KUKA KRL program: f1_Kuka_APT216T02S16.SRC

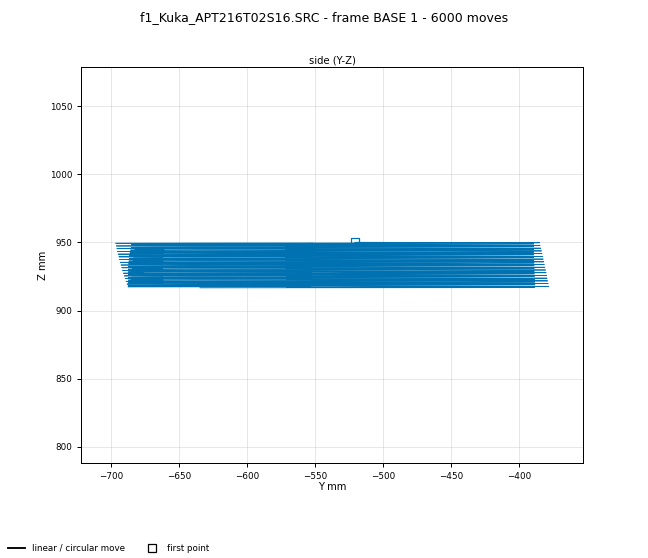
[picture p0: tool path of f1_Kuka_APT216T02S16.SRC in frame BASE 1, 6000 of 6001 moves have a stored position in this frame; points joined in program order, loops and branches not executed]
&ACCESS RVP
&REL 2
&PARAM TEMPLATE = C:\KRC\Roboter\Template\vorgabe
&PARAM EDITMASK = *
DEF f1_Kuka_APT216T02S16()


;FOLD INI;%{PE}%V3.2.0,%MKUKATPBASIS,%CINIT,%VCOMMON,%P
  ;FOLD BAS INI;%{E}%V3.2.0,%MKUKATPBASIS,%CINIT,%VINIT,%P
    GLOBAL INTERRUPT DECL 3 WHEN $STOPMESS==TRUE DO IR_STOPM ( )
    INTERRUPT ON 3
    BAS (#INITMOV,0 )
  ;ENDFOLD (BAS INI)
  ;FOLD USER INI;%{E}%V3.2.0,%MKUKATPUSER,%CINIT,%VINIT,%P
    ;Make your modifications here
  ;ENDFOLD (USER INI)
;ENDFOLD (INI)


;*** Make Null PTP Move
  PTP $pos_act

;*** Auto Load The Correct TOOL Data
  $tool=tool_data[2]

;*** Auto Load The Correct BASE Data
  $base=base_data[1]

  $ADVANCE = 5

;*** Restate Last Velocity
MMPM(30000.0)
SetRPM(8000)
LIN {X -0.232,Y -520.654,Z 950.174,A 0.000,B 0.000,C 90.000,E1 247.358} C_DIS
LIN {X 0.026,Y -518.514,Z 950.166,A 0.000,B 0.000,C 90.000,E1 245.869} C_DIS
LIN {X -0.020,Y -516.184,Z 950.158,A 0.000,B 0.000,C 90.000,E1 244.409} C_DIS
LIN {X -0.107,Y -513.864,Z 950.150,A 0.000,B 0.000,C 90.000,E1 242.948} C_DIS
LIN {X 0.234,Y -511.517,Z 950.141,A 0.000,B 0.000,C 90.000,E1 241.435} C_DIS
LIN {X 0.205,Y -509.572,Z 950.135,A 0.000,B 0.000,C 90.000,E1 240.255} C_DIS
LIN {X 0.092,Y -506.285,Z 950.125,A 0.000,B 0.000,C 90.000,E1 238.486} C_DIS
LIN {X 0.112,Y -503.056,Z 950.117,A 0.000,B 0.000,C 90.000,E1 236.993} C_DIS
LIN {X 0.178,Y -501.061,Z 950.112,A 0.000,B 0.000,C 90.000,E1 236.087} C_DIS
LIN {X -0.027,Y -497.587,Z 950.103,A 0.000,B 0.000,C 90.000,E1 234.609} C_DIS
LIN {X 0.259,Y -493.589,Z 950.093,A 0.000,B 0.000,C 90.000,E1 232.763} C_DIS
LIN {X 0.052,Y -489.488,Z 950.083,A 0.000,B 0.000,C 90.000,E1 230.964} C_DIS
LIN {X 0.021,Y -486.732,Z 950.076,A 0.000,B 0.000,C 90.000,E1 229.747} C_DIS
LIN {X -0.091,Y -482.456,Z 950.066,A 0.000,B 0.000,C 90.000,E1 227.919} C_DIS
LIN {X 0.103,Y -479.665,Z 950.059,A 0.000,B 0.000,C 90.000,E1 226.662} C_DIS
LIN {X 0.030,Y -476.272,Z 950.051,A 0.000,B 0.000,C 90.000,E1 225.121} C_DIS
LIN {X 0.084,Y -471.433,Z 950.039,A 0.000,B 0.000,C 90.000,E1 222.933} C_DIS
LIN {X -0.058,Y -467.344,Z 950.028,A 0.000,B 0.000,C 90.000,E1 221.067} C_DIS
LIN {X 0.155,Y -462.471,Z 950.016,A 0.000,B 0.000,C 90.000,E1 218.830} C_DIS
LIN {X 0.184,Y -459.007,Z 950.007,A 0.000,B 0.000,C 90.000,E1 217.237} C_DIS
LIN {X -0.125,Y -455.441,Z 949.998,A 0.000,B 0.000,C 90.000,E1 215.678} C_DIS
LIN {X 0.009,Y -449.781,Z 949.984,A 0.000,B 0.000,C 90.000,E1 213.086} C_DIS
LIN {X 0.154,Y -444.840,Z 949.971,A 0.000,B 0.000,C 90.000,E1 210.797} C_DIS
LIN {X -0.239,Y -439.153,Z 949.957,A 0.000,B 0.000,C 90.000,E1 208.231} C_DIS
LIN {X 0.100,Y -435.552,Z 949.948,A 0.000,B 0.000,C 90.000,E1 206.539} C_DIS
LIN {X -0.026,Y -431.162,Z 949.937,A 0.000,B 0.000,C 90.000,E1 204.567} C_DIS
LIN {X -0.015,Y -427.440,Z 949.927,A 0.000,B 0.000,C 90.000,E1 202.898} C_DIS
LIN {X 0.051,Y -420.044,Z 949.909,A 0.000,B 0.000,C 90.000,E1 199.523} C_DIS
LIN {X 0.037,Y -414.488,Z 949.893,A 0.000,B 0.000,C 90.000,E1 196.804} C_DIS
LIN {X 0.119,Y -411.074,Z 949.884,A 0.000,B 0.000,C 90.000,E1 195.079} C_DIS
LIN {X 0.127,Y -407.583,Z 949.874,A 0.000,B 0.000,C 90.000,E1 193.355} C_DIS
LIN {X -0.124,Y -404.196,Z 949.865,A 0.000,B 0.000,C 90.000,E1 191.658} C_DIS
LIN {X -0.050,Y -400.223,Z 949.853,A 0.000,B 0.000,C 90.000,E1 189.557} C_DIS
LIN {X -0.126,Y -396.847,Z 949.843,A 0.000,B 0.000,C 90.000,E1 187.814} C_DIS
LIN {X -0.021,Y -392.894,Z 949.832,A 0.000,B 0.000,C 90.000,E1 185.682} C_DIS
LIN {X -0.136,Y -388.562,Z 949.818,A 0.000,B 0.000,C 90.000,E1 183.212} C_DIS
LIN {X -0.091,Y -386.475,Z 949.810,A 0.000,B 0.000,C 90.000,E1 181.776} C_DIS
LIN {X 0.097,Y -385.701,Z 949.806,A 0.000,B 0.000,C 90.000,E1 181.031} C_DIS
LIN {X -0.107,Y -385.124,Z 949.802,A 0.000,B 0.000,C 90.000,E1 180.344} C_DIS
LIN {X 0.070,Y -384.918,Z 949.798,A 0.000,B 0.000,C 90.000,E1 179.599} C_DIS
LIN {X -0.140,Y -385.366,Z 949.794,A 0.000,B 0.000,C 90.000,E1 178.912} C_DIS
LIN {X 0.139,Y -385.840,Z 949.792,A 0.000,B 0.000,C 90.000,E1 178.511} C_DIS
LIN {X -0.006,Y -387.644,Z 949.788,A 0.000,B 0.000,C 90.000,E1 177.822} C_DIS
LIN {X 0.030,Y -388.934,Z 949.786,A 0.000,B 0.000,C 90.000,E1 177.478} C_DIS
LIN {X -0.113,Y -391.892,Z 949.783,A 0.000,B 0.000,C 90.000,E1 176.963} C_DIS
LIN {X 0.023,Y -394.043,Z 949.781,A 0.000,B 0.000,C 90.000,E1 176.617} C_DIS
LIN {X 0.167,Y -400.184,Z 949.778,A 0.000,B 0.000,C 90.000,E1 175.931} C_DIS
LIN {X -0.027,Y -406.077,Z 949.775,A 0.000,B 0.000,C 90.000,E1 175.412} C_DIS
LIN {X -0.026,Y -413.655,Z 949.771,A 0.000,B 0.000,C 90.000,E1 174.780} C_DIS
LIN {X 0.081,Y -421.495,Z 949.767,A 0.000,B 0.000,C 90.000,E1 174.090} C_DIS
LIN {X 0.102,Y -427.662,Z 949.764,A 0.000,B 0.000,C 90.000,E1 173.571} C_DIS
LIN {X 0.097,Y -436.825,Z 949.760,A 0.000,B 0.000,C 90.000,E1 172.761} C_DIS
LIN {X 0.074,Y -445.937,Z 949.755,A 0.000,B 0.000,C 90.000,E1 171.951} C_DIS
LIN {X -0.171,Y -455.808,Z 949.750,A 0.000,B 0.000,C 90.000,E1 171.027} C_DIS
LIN {X -0.006,Y -464.376,Z 949.745,A 0.000,B 0.000,C 90.000,E1 170.151} C_DIS
LIN {X 0.064,Y -469.840,Z 949.742,A 0.000,B 0.000,C 90.000,E1 169.567} C_DIS
LIN {X -0.010,Y -479.127,Z 949.736,A 0.000,B 0.000,C 90.000,E1 168.522} C_DIS
LIN {X -0.243,Y -484.228,Z 949.733,A 0.000,B 0.000,C 90.000,E1 167.937} C_DIS
LIN {X -0.041,Y -491.571,Z 949.728,A 0.000,B 0.000,C 90.000,E1 166.992} C_DIS
LIN {X 0.135,Y -498.521,Z 949.723,A 0.000,B 0.000,C 90.000,E1 166.061} C_DIS
LIN {X 0.092,Y -502.956,Z 949.719,A 0.000,B 0.000,C 90.000,E1 165.463} C_DIS
LIN {X 0.029,Y -509.105,Z 949.714,A 0.000,B 0.000,C 90.000,E1 164.574} C_DIS
LIN {X -0.123,Y -514.206,Z 949.710,A 0.000,B 0.000,C 90.000,E1 163.850} C_DIS
LIN {X 0.119,Y -518.896,Z 949.706,A 0.000,B 0.000,C 90.000,E1 163.087} C_DIS
LIN {X -0.265,Y -522.682,Z 949.703,A 0.000,B 0.000,C 90.000,E1 162.543} C_DIS
LIN {X 0.044,Y -529.996,Z 949.696,A 0.000,B 0.000,C 90.000,E1 161.348} C_DIS
LIN {X -0.016,Y -538.070,Z 949.689,A 0.000,B 0.000,C 90.000,E1 160.061} C_DIS
LIN {X -0.272,Y -541.475,Z 949.686,A 0.000,B 0.000,C 90.000,E1 159.518} C_DIS
LIN {X 0.310,Y -547.494,Z 949.681,A 0.000,B 0.000,C 90.000,E1 158.465} C_DIS
LIN {X 0.147,Y -554.103,Z 949.674,A 0.000,B 0.000,C 90.000,E1 157.358} C_DIS
LIN {X -0.117,Y -559.603,Z 949.669,A 0.000,B 0.000,C 90.000,E1 156.410} C_DIS
LIN {X -0.116,Y -563.343,Z 949.665,A 0.000,B 0.000,C 90.000,E1 155.717} C_DIS
LIN {X -0.015,Y -570.364,Z 949.657,A 0.000,B 0.000,C 90.000,E1 154.332} C_DIS
LIN {X -0.318,Y -576.661,Z 949.650,A 0.000,B 0.000,C 90.000,E1 152.999} C_DIS
LIN {X -0.126,Y -581.411,Z 949.644,A 0.000,B 0.000,C 90.000,E1 151.897} C_DIS
LIN {X 0.132,Y -585.685,Z 949.638,A 0.000,B 0.000,C 90.000,E1 150.795} C_DIS
LIN {X 0.172,Y -587.827,Z 949.635,A 0.000,B 0.000,C 90.000,E1 150.255} C_DIS
LIN {X -0.108,Y -592.795,Z 949.628,A 0.000,B 0.000,C 90.000,E1 148.948} C_DIS
LIN {X 0.310,Y -597.477,Z 949.620,A 0.000,B 0.000,C 90.000,E1 147.582} C_DIS
LIN {X 0.231,Y -602.930,Z 949.611,A 0.000,B 0.000,C 90.000,E1 146.008} C_DIS
LIN {X 0.070,Y -606.499,Z 949.606,A 0.000,B 0.000,C 90.000,E1 144.975} C_DIS
LIN {X 0.016,Y -611.876,Z 949.597,A 0.000,B 0.000,C 90.000,E1 143.417} C_DIS
LIN {X 0.061,Y -617.117,Z 949.588,A 0.000,B 0.000,C 90.000,E1 141.859} C_DIS
LIN {X 0.176,Y -621.563,Z 949.581,A 0.000,B 0.000,C 90.000,E1 140.561} C_DIS
LIN {X 0.025,Y -632.173,Z 949.564,A 0.000,B 0.000,C 90.000,E1 137.514} C_DIS
LIN {X 0.159,Y -634.999,Z 949.560,A 0.000,B 0.000,C 90.000,E1 136.743} C_DIS
LIN {X 0.041,Y -640.541,Z 949.551,A 0.000,B 0.000,C 90.000,E1 135.243} C_DIS
LIN {X 0.033,Y -646.038,Z 949.543,A 0.000,B 0.000,C 90.000,E1 133.743} C_DIS
LIN {X 0.086,Y -652.493,Z 949.533,A 0.000,B 0.000,C 90.000,E1 132.000} C_DIS
LIN {X -0.171,Y -658.949,Z 949.524,A 0.000,B 0.000,C 90.000,E1 130.297} C_DIS
LIN {X -0.190,Y -664.562,Z 949.516,A 0.000,B 0.000,C 90.000,E1 128.830} C_DIS
LIN {X -0.097,Y -670.115,Z 949.508,A 0.000,B 0.000,C 90.000,E1 127.363} C_DIS
LIN {X 0.112,Y -673.593,Z 949.502,A 0.000,B 0.000,C 90.000,E1 126.377} C_DIS
LIN {X -0.178,Y -676.931,Z 949.497,A 0.000,B 0.000,C 90.000,E1 125.438} C_DIS
LIN {X 0.289,Y -680.765,Z 949.490,A 0.000,B 0.000,C 90.000,E1 124.199} C_DIS
LIN {X -0.119,Y -684.239,Z 949.484,A 0.000,B 0.000,C 90.000,E1 123.038} C_DIS
LIN {X -0.102,Y -686.803,Z 949.478,A 0.000,B 0.000,C 90.000,E1 122.084} C_DIS
LIN {X -0.055,Y -689.089,Z 949.473,A 0.000,B 0.000,C 90.000,E1 121.131} C_DIS
LIN {X -0.200,Y -690.201,Z 949.470,A 0.000,B 0.000,C 90.000,E1 120.669} C_DIS
LIN {X -0.125,Y -692.059,Z 949.465,A 0.000,B 0.000,C 90.000,E1 119.716} C_DIS
LIN {X 0.229,Y -693.569,Z 949.460,A 0.000,B 0.000,C 90.000,E1 118.743} C_DIS
LIN {X 0.031,Y -694.577,Z 949.456,A 0.000,B 0.000,C 90.000,E1 118.052} C_DIS
LIN {X -0.189,Y -695.499,Z 949.451,A 0.000,B 0.000,C 90.000,E1 117.129} C_DIS
LIN {X -0.098,Y -696.065,Z 949.445,A 0.000,B 0.000,C 90.000,E1 116.181} C_DIS
LIN {X -0.364,Y -696.413,Z 949.439,A 0.000,B 0.000,C 90.000,E1 115.027} C_DIS
LIN {X 0.119,Y -696.392,Z 949.435,A 0.000,B 0.000,C 90.000,E1 114.283} C_DIS
LIN {X -0.005,Y -696.185,Z 949.432,A 0.000,B 0.000,C 90.000,E1 113.823} C_DIS
LIN {X 0.224,Y -695.279,Z 949.430,A 0.000,B 0.000,C 90.000,E1 113.334} C_DIS
LIN {X -0.165,Y -694.668,Z 949.428,A 0.000,B 0.000,C 90.000,E1 113.131} C_DIS
LIN {X -0.066,Y -692.739,Z 949.427,A 0.000,B 0.000,C 90.000,E1 112.770} C_DIS
LIN {X 0.174,Y -691.341,Z 949.425,A 0.000,B 0.000,C 90.000,E1 112.514} C_DIS
LIN {X 0.029,Y -690.332,Z 949.425,A 0.000,B 0.000,C 90.000,E1 112.408} C_DIS
LIN {X 0.145,Y -688.808,Z 949.424,A 0.000,B 0.000,C 90.000,E1 112.280} C_DIS
LIN {X -0.266,Y -683.650,Z 949.422,A 0.000,B 0.000,C 90.000,E1 112.025} C_DIS
LIN {X -0.132,Y -681.695,Z 949.422,A 0.000,B 0.000,C 90.000,E1 111.897} C_DIS
LIN {X -0.112,Y -676.345,Z 949.421,A 0.000,B 0.000,C 90.000,E1 111.716} C_DIS
LIN {X -0.005,Y -673.275,Z 949.420,A 0.000,B 0.000,C 90.000,E1 111.663} C_DIS
LIN {X 0.233,Y -667.551,Z 949.420,A 0.000,B 0.000,C 90.000,E1 111.589} C_DIS
LIN {X 0.175,Y -634.091,Z 949.420,A 0.000,B 0.000,C 90.000,E1 111.589} C_DIS
LIN {X 0.193,Y -629.702,Z 949.420,A 0.000,B 0.000,C 90.000,E1 111.535} C_DIS
LIN {X 0.223,Y -622.529,Z 949.419,A 0.000,B 0.000,C 90.000,E1 111.408} C_DIS
LIN {X 0.174,Y -615.532,Z 949.418,A 0.000,B 0.000,C 90.000,E1 111.227} C_DIS
LIN {X 0.223,Y -608.532,Z 949.417,A 0.000,B 0.000,C 90.000,E1 110.972} C_DIS
LIN {X -0.059,Y -600.335,Z 949.414,A 0.000,B 0.000,C 90.000,E1 110.610} C_DIS
LIN {X 0.310,Y -593.030,Z 949.412,A 0.000,B 0.000,C 90.000,E1 110.120} C_DIS
LIN {X -0.139,Y -577.483,Z 949.406,A 0.000,B 0.000,C 90.000,E1 109.033} C_DIS
LIN {X -0.162,Y -574.078,Z 949.405,A 0.000,B 0.000,C 90.000,E1 108.833} C_DIS
LIN {X -0.024,Y -569.119,Z 949.403,A 0.000,B 0.000,C 90.000,E1 108.544} C_DIS
LIN {X -0.086,Y -563.607,Z 949.402,A 0.000,B 0.000,C 90.000,E1 108.290} C_DIS
LIN {X 0.267,Y -555.303,Z 949.399,A 0.000,B 0.000,C 90.000,E1 107.873} C_DIS
LIN {X 0.222,Y -553.260,Z 949.399,A 0.000,B 0.000,C 90.000,E1 107.764} C_DIS
LIN {X -0.084,Y -551.662,Z 949.398,A 0.000,B 0.000,C 90.000,E1 107.638} C_DIS
LIN {X -0.137,Y -551.620,Z 949.398,A 0.000,B 0.000,C 90.000,E1 107.638} C_DIS
LIN {X -0.215,Y -551.221,Z 949.397,A 0.000,B 0.000,C 90.000,E1 107.457} C_DIS
LIN {X -0.144,Y -551.117,Z 949.395,A 0.000,B 0.000,C 90.000,E1 107.149} C_DIS
LIN {X 0.261,Y -551.695,Z 949.386,A 0.000,B 0.000,C 90.000,E1 105.426} C_DIS
LIN {X -0.161,Y -552.767,Z 949.373,A 0.000,B 0.000,C 90.000,E1 103.231} C_DIS
LIN {X -0.023,Y -554.814,Z 949.358,A 0.000,B 0.000,C 90.000,E1 100.423} C_DIS
LIN {X -0.026,Y -556.065,Z 949.350,A 0.000,B 0.000,C 90.000,E1 99.029} C_DIS
LIN {X -0.086,Y -557.277,Z 949.342,A 0.000,B 0.000,C 90.000,E1 97.644} C_DIS
LIN {X -0.187,Y -558.194,Z 949.336,A 0.000,B 0.000,C 90.000,E1 96.543} C_DIS
LIN {X 0.212,Y -558.934,Z 949.330,A 0.000,B 0.000,C 90.000,E1 95.391} C_DIS
LIN {X 0.018,Y -559.641,Z 949.324,A 0.000,B 0.000,C 90.000,E1 94.302} C_DIS
LIN {X 0.054,Y -560.601,Z 949.315,A 0.000,B 0.000,C 90.000,E1 92.636} C_DIS
LIN {X -0.113,Y -561.108,Z 949.309,A 0.000,B 0.000,C 90.000,E1 91.547} C_DIS
LIN {X -0.190,Y -561.700,Z 949.301,A 0.000,B 0.000,C 90.000,E1 90.172} C_DIS
LIN {X 0.207,Y -562.043,Z 949.295,A 0.000,B 0.000,C 90.000,E1 89.026} C_DIS
LIN {X 0.161,Y -562.350,Z 949.287,A 0.000,B 0.000,C 90.000,E1 87.650} C_DIS
LIN {X 0.120,Y -562.635,Z 949.279,A 0.000,B 0.000,C 90.000,E1 86.274} C_DIS
LIN {X 0.210,Y -562.883,Z 949.270,A 0.000,B 0.000,C 90.000,E1 84.609} C_DIS
LIN {X -0.140,Y -563.149,Z 949.261,A 0.000,B 0.000,C 90.000,E1 82.989} C_DIS
LIN {X -0.072,Y -563.754,Z 949.247,A 0.000,B 0.000,C 90.000,E1 80.500} C_DIS
LIN {X 0.032,Y -564.679,Z 949.235,A 0.000,B 0.000,C 90.000,E1 78.285} C_DIS
LIN {X -0.287,Y -565.934,Z 949.223,A 0.000,B 0.000,C 90.000,E1 76.117} C_DIS
LIN {X -0.089,Y -566.976,Z 949.214,A 0.000,B 0.000,C 90.000,E1 74.448} C_DIS
LIN {X 0.136,Y -568.043,Z 949.204,A 0.000,B 0.000,C 90.000,E1 72.779} C_DIS
LIN {X 0.207,Y -568.808,Z 949.197,A 0.000,B 0.000,C 90.000,E1 71.402} C_DIS
LIN {X -0.066,Y -569.546,Z 949.189,A 0.000,B 0.000,C 90.000,E1 70.061} C_DIS
LIN {X 0.020,Y -570.119,Z 949.180,A 0.000,B 0.000,C 90.000,E1 68.411} C_DIS
LIN {X -0.202,Y -570.590,Z 949.171,A 0.000,B 0.000,C 90.000,E1 66.794} C_DIS
LIN {X 0.170,Y -571.025,Z 949.160,A 0.000,B 0.000,C 90.000,E1 64.845} C_DIS
LIN {X 0.192,Y -571.266,Z 949.151,A 0.000,B 0.000,C 90.000,E1 63.204} C_DIS
LIN {X 0.125,Y -571.435,Z 949.144,A 0.000,B 0.000,C 90.000,E1 61.847} C_DIS
LIN {X 0.165,Y -571.468,Z 949.135,A 0.000,B 0.000,C 90.000,E1 60.205} C_DIS
LIN {X 0.008,Y -571.634,Z 949.126,A 0.000,B 0.000,C 90.000,E1 58.584} C_DIS
LIN {X -0.266,Y -571.503,Z 949.118,A 0.000,B 0.000,C 90.000,E1 57.248} C_DIS
LIN {X -0.244,Y -571.139,Z 949.110,A 0.000,B 0.000,C 90.000,E1 55.881} C_DIS
LIN {X 0.092,Y -570.671,Z 949.103,A 0.000,B 0.000,C 90.000,E1 54.482} C_DIS
LIN {X 0.357,Y -570.473,Z 949.100,A 0.000,B 0.000,C 90.000,E1 53.909} C_DIS
LIN {X -0.045,Y -569.986,Z 949.095,A 0.000,B 0.000,C 90.000,E1 53.130} C_DIS
LIN {X 0.024,Y -569.081,Z 949.089,A 0.000,B 0.000,C 90.000,E1 52.029} C_DIS
LIN {X 0.085,Y -568.018,Z 949.083,A 0.000,B 0.000,C 90.000,E1 50.928} C_DIS
LIN {X 0.010,Y -567.101,Z 949.078,A 0.000,B 0.000,C 90.000,E1 50.114} C_DIS
LIN {X -0.077,Y -566.046,Z 949.074,A 0.000,B 0.000,C 90.000,E1 49.299} C_DIS
LIN {X -0.181,Y -564.794,Z 949.069,A 0.000,B 0.000,C 90.000,E1 48.485} C_DIS
LIN {X -0.248,Y -562.711,Z 949.063,A 0.000,B 0.000,C 90.000,E1 47.391} C_DIS
LIN {X -0.098,Y -561.646,Z 949.060,A 0.000,B 0.000,C 90.000,E1 46.824} C_DIS
LIN {X 0.122,Y -559.750,Z 949.056,A 0.000,B 0.000,C 90.000,E1 45.972} C_DIS
LIN {X -0.081,Y -557.570,Z 949.051,A 0.000,B 0.000,C 90.000,E1 45.162} C_DIS
LIN {X 0.034,Y -556.031,Z 949.048,A 0.000,B 0.000,C 90.000,E1 44.595} C_DIS
LIN {X -0.207,Y -553.337,Z 949.043,A 0.000,B 0.000,C 90.000,E1 43.785} C_DIS
LIN {X -0.125,Y -551.495,Z 949.040,A 0.000,B 0.000,C 90.000,E1 43.218} C_DIS
LIN {X -0.017,Y -548.288,Z 949.035,A 0.000,B 0.000,C 90.000,E1 42.366} C_DIS
LIN {X 0.056,Y -544.757,Z 949.031,A 0.000,B 0.000,C 90.000,E1 41.515} C_DIS
LIN {X 0.281,Y -542.809,Z 949.028,A 0.000,B 0.000,C 90.000,E1 41.067} C_DIS
LIN {X -0.064,Y -538.565,Z 949.024,A 0.000,B 0.000,C 90.000,E1 40.253} C_DIS
LIN {X -0.279,Y -534.725,Z 949.020,A 0.000,B 0.000,C 90.000,E1 39.564} C_DIS
LIN {X 0.043,Y -529.767,Z 949.015,A 0.000,B 0.000,C 90.000,E1 38.669} C_DIS
LIN {X 0.122,Y -523.679,Z 949.009,A 0.000,B 0.000,C 90.000,E1 37.649} C_DIS
LIN {X 0.041,Y -520.035,Z 949.006,A 0.000,B 0.000,C 90.000,E1 37.076} C_DIS
LIN {X -0.312,Y -513.139,Z 949.000,A 0.000,B 0.000,C 90.000,E1 36.091} C_DIS
LIN {X 0.055,Y -507.914,Z 948.996,A 0.000,B 0.000,C 90.000,E1 35.311} C_DIS
LIN {X -0.138,Y -503.436,Z 948.993,A 0.000,B 0.000,C 90.000,E1 34.739} C_DIS
LIN {X -0.031,Y -499.916,Z 948.990,A 0.000,B 0.000,C 90.000,E1 34.278} C_DIS
LIN {X -0.079,Y -496.182,Z 948.988,A 0.000,B 0.000,C 90.000,E1 33.833} C_DIS
LIN {X -0.167,Y -488.144,Z 948.983,A 0.000,B 0.000,C 90.000,E1 32.959} C_DIS
LIN {X 0.054,Y -481.171,Z 948.979,A 0.000,B 0.000,C 90.000,E1 32.212} C_DIS
LIN {X -0.140,Y -475.423,Z 948.976,A 0.000,B 0.000,C 90.000,E1 31.671} C_DIS
LIN {X -0.059,Y -466.585,Z 948.971,A 0.000,B 0.000,C 90.000,E1 30.846} C_DIS
LIN {X -0.078,Y -459.131,Z 948.968,A 0.000,B 0.000,C 90.000,E1 30.178} C_DIS
LIN {X -0.255,Y -448.516,Z 948.963,A 0.000,B 0.000,C 90.000,E1 29.283} C_DIS
LIN {X -0.056,Y -428.627,Z 948.953,A 0.000,B 0.000,C 90.000,E1 27.564} C_DIS
LIN {X -0.085,Y -412.114,Z 948.945,A 0.000,B 0.000,C 90.000,E1 26.052} C_DIS
LIN {X 0.032,Y -400.392,Z 948.938,A 0.000,B 0.000,C 90.000,E1 24.847} C_DIS
LIN {X 0.149,Y -397.529,Z 948.936,A 0.000,B 0.000,C 90.000,E1 24.515} C_DIS
LIN {X -0.027,Y -394.399,Z 948.934,A 0.000,B 0.000,C 90.000,E1 24.131} C_DIS
LIN {X -0.152,Y -392.235,Z 948.932,A 0.000,B 0.000,C 90.000,E1 23.770} C_DIS
LIN {X 0.028,Y -391.305,Z 948.931,A 0.000,B 0.000,C 90.000,E1 23.567} C_DIS
LIN {X 0.111,Y -389.845,Z 948.928,A 0.000,B 0.000,C 90.000,E1 23.025} C_DIS
LIN {X -0.029,Y -389.162,Z 948.924,A 0.000,B 0.000,C 90.000,E1 22.333} C_DIS
LIN {X 0.201,Y -389.528,Z 948.919,A 0.000,B 0.000,C 90.000,E1 21.408} C_DIS
LIN {X 0.076,Y -393.067,Z 948.897,A 0.000,B 0.000,C 90.000,E1 17.511} C_DIS
LIN {X -0.181,Y -396.430,Z 948.882,A 0.000,B 0.000,C 90.000,E1 14.717} C_DIS
LIN {X -0.107,Y -399.795,Z 948.868,A 0.000,B 0.000,C 90.000,E1 12.243} C_DIS
LIN {X -0.097,Y -404.793,Z 948.851,A 0.000,B 0.000,C 90.000,E1 9.095} C_DIS
LIN {X -0.041,Y -410.390,Z 948.833,A 0.000,B 0.000,C 90.000,E1 5.967} C_DIS
LIN {X 0.057,Y -417.434,Z 948.814,A 0.000,B 0.000,C 90.000,E1 2.522} C_DIS
LIN {X 0.208,Y -424.749,Z 948.797,A 0.000,B 0.000,C 90.000,E1 359.427} C_DIS
LIN {X -0.167,Y -425.696,Z 948.795,A 0.000,B 0.000,C 90.000,E1 359.141} C_DIS
LIN {X -0.058,Y -428.393,Z 948.791,A 0.000,B 0.000,C 90.000,E1 358.453} C_DIS
LIN {X 0.090,Y -429.543,Z 948.790,A 0.000,B 0.000,C 90.000,E1 358.224} C_DIS
LIN {X 0.092,Y -431.486,Z 948.789,A 0.000,B 0.000,C 90.000,E1 357.936} C_DIS
LIN {X 0.216,Y -435.092,Z 948.786,A 0.000,B 0.000,C 90.000,E1 357.535} C_DIS
LIN {X 0.188,Y -440.022,Z 948.785,A 0.000,B 0.000,C 90.000,E1 357.192} C_DIS
LIN {X 0.066,Y -458.415,Z 948.779,A 0.000,B 0.000,C 90.000,E1 356.274} C_DIS
LIN {X -0.181,Y -466.700,Z 948.777,A 0.000,B 0.000,C 90.000,E1 355.869} C_DIS
LIN {X 0.094,Y -480.168,Z 948.773,A 0.000,B 0.000,C 90.000,E1 355.122} C_DIS
LIN {X 0.084,Y -491.926,Z 948.769,A 0.000,B 0.000,C 90.000,E1 354.489} C_DIS
LIN {X -0.062,Y -498.505,Z 948.768,A 0.000,B 0.000,C 90.000,E1 354.147} C_DIS
LIN {X 0.115,Y -507.951,Z 948.764,A 0.000,B 0.000,C 90.000,E1 353.571} C_DIS
LIN {X -0.046,Y -517.568,Z 948.761,A 0.000,B 0.000,C 90.000,E1 352.996} C_DIS
LIN {X 0.144,Y -526.710,Z 948.758,A 0.000,B 0.000,C 90.000,E1 352.356} C_DIS
LIN {X -0.198,Y -534.129,Z 948.755,A 0.000,B 0.000,C 90.000,E1 351.837} C_DIS
LIN {X -0.212,Y -541.363,Z 948.751,A 0.000,B 0.000,C 90.000,E1 351.254} C_DIS
LIN {X -0.050,Y -548.207,Z 948.748,A 0.000,B 0.000,C 90.000,E1 350.622} C_DIS
LIN {X -0.234,Y -554.623,Z 948.744,A 0.000,B 0.000,C 90.000,E1 349.982} C_DIS
LIN {X 0.135,Y -559.615,Z 948.741,A 0.000,B 0.000,C 90.000,E1 349.398} C_DIS
LIN {X 0.181,Y -565.330,Z 948.737,A 0.000,B 0.000,C 90.000,E1 348.701} C_DIS
LIN {X -0.037,Y -569.568,Z 948.734,A 0.000,B 0.000,C 90.000,E1 348.173} C_DIS
LIN {X 0.211,Y -574.517,Z 948.731,A 0.000,B 0.000,C 90.000,E1 347.465} C_DIS
LIN {X 0.273,Y -579.999,Z 948.726,A 0.000,B 0.000,C 90.000,E1 346.645} C_DIS
LIN {X 0.058,Y -586.520,Z 948.720,A 0.000,B 0.000,C 90.000,E1 345.589} C_DIS
LIN {X 0.307,Y -591.809,Z 948.715,A 0.000,B 0.000,C 90.000,E1 344.629} C_DIS
LIN {X -0.106,Y -596.683,Z 948.710,A 0.000,B 0.000,C 90.000,E1 343.740} C_DIS
LIN {X 0.047,Y -601.896,Z 948.704,A 0.000,B 0.000,C 90.000,E1 342.670} C_DIS
LIN {X 0.179,Y -608.028,Z 948.697,A 0.000,B 0.000,C 90.000,E1 341.348} C_DIS
LIN {X 0.085,Y -612.604,Z 948.691,A 0.000,B 0.000,C 90.000,E1 340.315} C_DIS
LIN {X 0.013,Y -617.926,Z 948.684,A 0.000,B 0.000,C 90.000,E1 339.028} C_DIS
LIN {X 0.275,Y -621.863,Z 948.678,A 0.000,B 0.000,C 90.000,E1 337.975} C_DIS
LIN {X 0.019,Y -625.619,Z 948.672,A 0.000,B 0.000,C 90.000,E1 336.975} C_DIS
LIN {X -0.165,Y -629.912,Z 948.665,A 0.000,B 0.000,C 90.000,E1 335.717} C_DIS
LIN {X 0.292,Y -633.837,Z 948.658,A 0.000,B 0.000,C 90.000,E1 334.409} C_DIS
LIN {X -0.057,Y -637.521,Z 948.651,A 0.000,B 0.000,C 90.000,E1 333.179} C_DIS
LIN {X 0.166,Y -640.207,Z 948.645,A 0.000,B 0.000,C 90.000,E1 332.153} C_DIS
LIN {X -0.146,Y -642.621,Z 948.640,A 0.000,B 0.000,C 90.000,E1 331.179} C_DIS
LIN {X -0.040,Y -645.468,Z 948.633,A 0.000,B 0.000,C 90.000,E1 329.921} C_DIS
LIN {X 0.114,Y -648.016,Z 948.626,A 0.000,B 0.000,C 90.000,E1 328.663} C_DIS
LIN {X -0.252,Y -650.147,Z 948.619,A 0.000,B 0.000,C 90.000,E1 327.454} C_DIS
LIN {X 0.229,Y -651.668,Z 948.614,A 0.000,B 0.000,C 90.000,E1 326.421} C_DIS
LIN {X 0.272,Y -653.310,Z 948.607,A 0.000,B 0.000,C 90.000,E1 325.182} C_DIS
LIN {X -0.195,Y -654.159,Z 948.603,A 0.000,B 0.000,C 90.000,E1 324.482} C_DIS
LIN {X -0.201,Y -655.114,Z 948.597,A 0.000,B 0.000,C 90.000,E1 323.497} C_DIS
LIN {X 0.204,Y -656.376,Z 948.589,A 0.000,B 0.000,C 90.000,E1 321.984} C_DIS
LIN {X 0.074,Y -657.682,Z 948.579,A 0.000,B 0.000,C 90.000,E1 320.275} C_DIS
LIN {X -0.029,Y -658.532,Z 948.573,A 0.000,B 0.000,C 90.000,E1 319.057} C_DIS
LIN {X -0.226,Y -660.444,Z 948.558,A 0.000,B 0.000,C 90.000,E1 316.377} C_DIS
LIN {X -0.304,Y -661.245,Z 948.552,A 0.000,B 0.000,C 90.000,E1 315.405} C_DIS
LIN {X 0.044,Y -663.106,Z 948.540,A 0.000,B 0.000,C 90.000,E1 313.176} C_DIS
LIN {X 0.021,Y -664.458,Z 948.532,A 0.000,B 0.000,C 90.000,E1 311.714} C_DIS
LIN {X 0.035,Y -665.578,Z 948.525,A 0.000,B 0.000,C 90.000,E1 310.496} C_DIS
LIN {X 0.059,Y -666.560,Z 948.518,A 0.000,B 0.000,C 90.000,E1 309.277} C_DIS
LIN {X -0.333,Y -667.496,Z 948.512,A 0.000,B 0.000,C 90.000,E1 308.096} C_DIS
LIN {X -0.251,Y -667.873,Z 948.509,A 0.000,B 0.000,C 90.000,E1 307.604} C_DIS
LIN {X -0.097,Y -668.375,Z 948.502,A 0.000,B 0.000,C 90.000,E1 306.377} C_DIS
LIN {X -0.235,Y -668.877,Z 948.493,A 0.000,B 0.000,C 90.000,E1 304.692} C_DIS
LIN {X 0.188,Y -669.527,Z 948.483,A 0.000,B 0.000,C 90.000,E1 302.959} C_DIS
LIN {X 0.253,Y -670.367,Z 948.474,A 0.000,B 0.000,C 90.000,E1 301.258} C_DIS
LIN {X 0.345,Y -674.131,Z 948.452,A 0.000,B 0.000,C 90.000,E1 297.385} C_DIS
LIN {X -0.410,Y -677.717,Z 948.440,A 0.000,B 0.000,C 90.000,E1 295.283} C_DIS
LIN {X -0.346,Y -679.725,Z 948.434,A 0.000,B 0.000,C 90.000,E1 294.079} C_DIS
LIN {X -0.032,Y -680.838,Z 948.430,A 0.000,B 0.000,C 90.000,E1 293.334} C_DIS
LIN {X -0.331,Y -681.524,Z 948.426,A 0.000,B 0.000,C 90.000,E1 292.642} C_DIS
LIN {X -0.194,Y -681.362,Z 948.423,A 0.000,B 0.000,C 90.000,E1 292.153} C_DIS
LIN {X 0.002,Y -681.134,Z 948.422,A 0.000,B 0.000,C 90.000,E1 291.897} C_DIS
LIN {X -0.056,Y -680.338,Z 948.420,A 0.000,B 0.000,C 90.000,E1 291.663} C_DIS
LIN {X 0.080,Y -678.053,Z 948.418,A 0.000,B 0.000,C 90.000,E1 291.173} C_DIS
LIN {X 0.172,Y -677.053,Z 948.417,A 0.000,B 0.000,C 90.000,E1 291.046} C_DIS
LIN {X -0.223,Y -674.434,Z 948.416,A 0.000,B 0.000,C 90.000,E1 290.844} C_DIS
LIN {X -0.077,Y -671.639,Z 948.414,A 0.000,B 0.000,C 90.000,E1 290.610} C_DIS
LIN {X -0.020,Y -666.907,Z 948.413,A 0.000,B 0.000,C 90.000,E1 290.301} C_DIS
LIN {X 0.227,Y -661.860,Z 948.411,A 0.000,B 0.000,C 90.000,E1 289.939} C_DIS
LIN {X -0.028,Y -660.825,Z 948.411,A 0.000,B 0.000,C 90.000,E1 289.885} C_DIS
LIN {X -0.096,Y -660.785,Z 948.410,A 0.000,B 0.000,C 90.000,E1 289.885} C_DIS
LIN {X 0.292,Y -660.270,Z 948.410,A 0.000,B 0.000,C 90.000,E1 289.758} C_DIS
LIN {X 0.225,Y -660.259,Z 948.410,A 0.000,B 0.000,C 90.000,E1 289.758} C_DIS
LIN {X 0.102,Y -660.344,Z 948.409,A 0.000,B 0.000,C 90.000,E1 289.523} C_DIS
LIN {X 0.125,Y -660.794,Z 948.408,A 0.000,B 0.000,C 90.000,E1 289.341} C_DIS
LIN {X 0.289,Y -662.012,Z 948.406,A 0.000,B 0.000,C 90.000,E1 288.960} C_DIS
LIN {X 0.086,Y -669.194,Z 948.398,A 0.000,B 0.000,C 90.000,E1 287.638} C_DIS
LIN {X -0.064,Y -671.729,Z 948.395,A 0.000,B 0.000,C 90.000,E1 287.166} C_DIS
LIN {X -0.064,Y -674.896,Z 948.391,A 0.000,B 0.000,C 90.000,E1 286.441} C_DIS
LIN {X -0.043,Y -677.464,Z 948.387,A 0.000,B 0.000,C 90.000,E1 285.717} C_DIS
LIN {X -0.138,Y -678.887,Z 948.385,A 0.000,B 0.000,C 90.000,E1 285.245} C_DIS
LIN {X -0.262,Y -680.604,Z 948.381,A 0.000,B 0.000,C 90.000,E1 284.537} C_DIS
LIN {X 0.296,Y -681.962,Z 948.377,A 0.000,B 0.000,C 90.000,E1 283.772} C_DIS
LIN {X 0.206,Y -683.143,Z 948.373,A 0.000,B 0.000,C 90.000,E1 283.063} C_DIS
LIN {X 0.124,Y -684.038,Z 948.369,A 0.000,B 0.000,C 90.000,E1 282.355} C_DIS
LIN {X -0.095,Y -684.630,Z 948.365,A 0.000,B 0.000,C 90.000,E1 281.658} C_DIS
LIN {X -0.144,Y -684.816,Z 948.362,A 0.000,B 0.000,C 90.000,E1 281.186} C_DIS
LIN {X -0.197,Y -684.693,Z 948.359,A 0.000,B 0.000,C 90.000,E1 280.715} C_DIS
LIN {X 0.297,Y -684.272,Z 948.357,A 0.000,B 0.000,C 90.000,E1 280.197} C_DIS
LIN {X 0.236,Y -683.453,Z 948.354,A 0.000,B 0.000,C 90.000,E1 279.726} C_DIS
LIN {X 0.054,Y -682.344,Z 948.352,A 0.000,B 0.000,C 90.000,E1 279.265} C_DIS
LIN {X 0.016,Y -681.735,Z 948.350,A 0.000,B 0.000,C 90.000,E1 279.029} C_DIS
LIN {X -0.173,Y -680.105,Z 948.348,A 0.000,B 0.000,C 90.000,E1 278.568} C_DIS
LIN {X 0.247,Y -677.032,Z 948.344,A 0.000,B 0.000,C 90.000,E1 277.814} C_DIS
LIN {X -0.122,Y -673.513,Z 948.340,A 0.000,B 0.000,C 90.000,E1 277.125} C_DIS
LIN {X -0.274,Y -671.594,Z 948.338,A 0.000,B 0.000,C 90.000,E1 276.777} C_DIS
LIN {X 0.143,Y -668.794,Z 948.335,A 0.000,B 0.000,C 90.000,E1 276.258} C_DIS
LIN {X -0.125,Y -665.751,Z 948.332,A 0.000,B 0.000,C 90.000,E1 275.796} C_DIS
LIN {X 0.158,Y -661.292,Z 948.329,A 0.000,B 0.000,C 90.000,E1 275.163} C_DIS
LIN {X -0.119,Y -658.439,Z 948.327,A 0.000,B 0.000,C 90.000,E1 274.821} C_DIS
LIN {X 0.001,Y -651.781,Z 948.323,A 0.000,B 0.000,C 90.000,E1 274.073} C_DIS
LIN {X 0.272,Y -647.055,Z 948.320,A 0.000,B 0.000,C 90.000,E1 273.555} C_DIS
LIN {X -0.012,Y -642.044,Z 948.317,A 0.000,B 0.000,C 90.000,E1 273.094} C_DIS
LIN {X -0.136,Y -636.787,Z 948.315,A 0.000,B 0.000,C 90.000,E1 272.636} C_DIS
LIN {X -0.096,Y -631.333,Z 948.312,A 0.000,B 0.000,C 90.000,E1 272.178} C_DIS
LIN {X -0.280,Y -624.030,Z 948.309,A 0.000,B 0.000,C 90.000,E1 271.661} C_DIS
LIN {X -0.077,Y -616.380,Z 948.306,A 0.000,B 0.000,C 90.000,E1 271.146} C_DIS
LIN {X 0.116,Y -610.051,Z 948.304,A 0.000,B 0.000,C 90.000,E1 270.745} C_DIS
LIN {X -0.017,Y -603.473,Z 948.302,A 0.000,B 0.000,C 90.000,E1 270.401} C_DIS
LIN {X -0.235,Y -598.439,Z 948.301,A 0.000,B 0.000,C 90.000,E1 270.172} C_DIS
LIN {X 0.160,Y -591.399,Z 948.299,A 0.000,B 0.000,C 90.000,E1 269.828} C_DIS
LIN {X 0.278,Y -584.013,Z 948.298,A 0.000,B 0.000,C 90.000,E1 269.542} C_DIS
LIN {X 0.234,Y -578.151,Z 948.297,A 0.000,B 0.000,C 90.000,E1 269.370} C_DIS
LIN {X 0.080,Y -570.455,Z 948.296,A 0.000,B 0.000,C 90.000,E1 269.198} C_DIS
LIN {X 0.056,Y -564.645,Z 948.295,A 0.000,B 0.000,C 90.000,E1 269.083} C_DIS
LIN {X -0.096,Y -558.396,Z 948.295,A 0.000,B 0.000,C 90.000,E1 269.026} C_DIS
LIN {X 0.014,Y -550.975,Z 948.294,A 0.000,B 0.000,C 90.000,E1 268.969} C_DIS
LIN {X 0.200,Y -548.037,Z 948.294,A 0.000,B 0.000,C 90.000,E1 268.912} C_DIS
LIN {X 0.125,Y -543.889,Z 948.293,A 0.000,B 0.000,C 90.000,E1 268.682} C_DIS
LIN {X 0.071,Y -543.819,Z 948.293,A 0.000,B 0.000,C 90.000,E1 268.682} C_DIS
LIN {X -0.084,Y -543.151,Z 948.291,A 0.000,B 0.000,C 90.000,E1 268.396} C_DIS
LIN {X -0.263,Y -542.588,Z 948.287,A 0.000,B 0.000,C 90.000,E1 267.707} C_DIS
LIN {X 0.036,Y -540.539,Z 948.273,A 0.000,B 0.000,C 90.000,E1 265.122} C_DIS
LIN {X 0.183,Y -539.538,Z 948.265,A 0.000,B 0.000,C 90.000,E1 263.685} C_DIS
LIN {X -0.107,Y -538.365,Z 948.256,A 0.000,B 0.000,C 90.000,E1 262.008} C_DIS
LIN {X 0.006,Y -537.683,Z 948.251,A 0.000,B 0.000,C 90.000,E1 261.141} C_DIS
LIN {X 0.134,Y -537.129,Z 948.248,A 0.000,B 0.000,C 90.000,E1 260.557} C_DIS
LIN {X -0.242,Y -535.680,Z 948.241,A 0.000,B 0.000,C 90.000,E1 259.454} C_DIS
LIN {X 0.184,Y -532.678,Z 948.229,A 0.000,B 0.000,C 90.000,E1 257.117} C_DIS
LIN {X 0.208,Y -530.309,Z 948.217,A 0.000,B 0.000,C 90.000,E1 255.102} C_DIS
LIN {X 0.150,Y -528.327,Z 948.208,A 0.000,B 0.000,C 90.000,E1 253.378} C_DIS
LIN {X 0.029,Y -526.643,Z 948.200,A 0.000,B 0.000,C 90.000,E1 251.945} C_DIS
LIN {X 0.030,Y -524.792,Z 948.192,A 0.000,B 0.000,C 90.000,E1 250.496} C_DIS
LIN {X 0.172,Y -522.925,Z 948.184,A 0.000,B 0.000,C 90.000,E1 249.028} C_DIS
LIN {X -0.008,Y -521.074,Z 948.176,A 0.000,B 0.000,C 90.000,E1 247.592} C_DIS
LIN {X 0.265,Y -518.975,Z 948.167,A 0.000,B 0.000,C 90.000,E1 246.102} C_DIS
LIN {X 0.015,Y -516.639,Z 948.159,A 0.000,B 0.000,C 90.000,E1 244.665} C_DIS
LIN {X -0.064,Y -514.310,Z 948.151,A 0.000,B 0.000,C 90.000,E1 243.204} C_DIS
LIN {X 0.042,Y -511.971,Z 948.143,A 0.000,B 0.000,C 90.000,E1 241.719} C_DIS
LIN {X -0.094,Y -509.560,Z 948.135,A 0.000,B 0.000,C 90.000,E1 240.255} C_DIS
LIN {X 0.060,Y -506.270,Z 948.125,A 0.000,B 0.000,C 90.000,E1 238.456} C_DIS
LIN {X 0.091,Y -503.025,Z 948.117,A 0.000,B 0.000,C 90.000,E1 236.962} C_DIS
LIN {X -0.116,Y -501.027,Z 948.112,A 0.000,B 0.000,C 90.000,E1 236.087} C_DIS
LIN {X -0.194,Y -498.233,Z 948.105,A 0.000,B 0.000,C 90.000,E1 234.895} C_DIS
LIN {X -0.033,Y -493.555,Z 948.093,A 0.000,B 0.000,C 90.000,E1 232.763} C_DIS
LIN {X 0.070,Y -489.459,Z 948.083,A 0.000,B 0.000,C 90.000,E1 230.928} C_DIS
LIN {X 0.103,Y -486.701,Z 948.076,A 0.000,B 0.000,C 90.000,E1 229.703} C_DIS
LIN {X 0.168,Y -483.155,Z 948.068,A 0.000,B 0.000,C 90.000,E1 228.162} C_DIS
LIN {X -0.056,Y -478.972,Z 948.057,A 0.000,B 0.000,C 90.000,E1 226.338} C_DIS
LIN {X 0.084,Y -476.245,Z 948.051,A 0.000,B 0.000,C 90.000,E1 225.081} C_DIS
LIN {X -0.198,Y -471.407,Z 948.038,A 0.000,B 0.000,C 90.000,E1 222.933} C_DIS
LIN {X -0.100,Y -468.017,Z 948.030,A 0.000,B 0.000,C 90.000,E1 221.353} C_DIS
LIN {X -0.122,Y -462.478,Z 948.016,A 0.000,B 0.000,C 90.000,E1 218.830} C_DIS
LIN {X -0.073,Y -458.286,Z 948.005,A 0.000,B 0.000,C 90.000,E1 216.916} C_DIS
LIN {X -0.033,Y -454.734,Z 947.996,A 0.000,B 0.000,C 90.000,E1 215.311} C_DIS
LIN {X 0.117,Y -449.802,Z 947.984,A 0.000,B 0.000,C 90.000,E1 213.038} C_DIS
LIN {X -0.048,Y -444.086,Z 947.969,A 0.000,B 0.000,C 90.000,E1 210.463} C_DIS
LIN {X 0.093,Y -439.152,Z 947.957,A 0.000,B 0.000,C 90.000,E1 208.153} C_DIS
LIN {X 0.055,Y -434.830,Z 947.946,A 0.000,B 0.000,C 90.000,E1 206.181} C_DIS
LIN {X 0.107,Y -431.133,Z 947.936,A 0.000,B 0.000,C 90.000,E1 204.515} C_DIS
LIN {X -0.271,Y -427.448,Z 947.927,A 0.000,B 0.000,C 90.000,E1 202.898} C_DIS
LIN {X 0.161,Y -420.781,Z 947.910,A 0.000,B 0.000,C 90.000,E1 199.812} C_DIS
LIN {X 0.156,Y -415.182,Z 947.895,A 0.000,B 0.000,C 90.000,E1 197.094} C_DIS
LIN {X -0.152,Y -411.752,Z 947.886,A 0.000,B 0.000,C 90.000,E1 195.426} C_DIS
LIN {X -0.133,Y -408.287,Z 947.876,A 0.000,B 0.000,C 90.000,E1 193.703} C_DIS
LIN {X 0.023,Y -404.862,Z 947.866,A 0.000,B 0.000,C 90.000,E1 191.951} C_DIS
LIN {X 0.113,Y -400.891,Z 947.855,A 0.000,B 0.000,C 90.000,E1 189.849} C_DIS
LIN {X 0.030,Y -396.832,Z 947.843,A 0.000,B 0.000,C 90.000,E1 187.757} C_DIS
LIN {X 0.135,Y -392.877,Z 947.831,A 0.000,B 0.000,C 90.000,E1 185.625} C_DIS
LIN {X 0.108,Y -389.090,Z 947.820,A 0.000,B 0.000,C 90.000,E1 183.498} C_DIS
LIN {X 0.062,Y -386.318,Z 947.810,A 0.000,B 0.000,C 90.000,E1 181.718} C_DIS
LIN {X -0.037,Y -385.836,Z 947.808,A 0.000,B 0.000,C 90.000,E1 181.375} C_DIS
LIN {X 0.042,Y -384.825,Z 947.802,A 0.000,B 0.000,C 90.000,E1 180.286} C_DIS
LIN {X -0.167,Y -384.535,Z 947.798,A 0.000,B 0.000,C 90.000,E1 179.599} C_DIS
LIN {X -0.169,Y -384.661,Z 947.796,A 0.000,B 0.000,C 90.000,E1 179.255} C_DIS
LIN {X 0.109,Y -384.610,Z 947.794,A 0.000,B 0.000,C 90.000,E1 178.854} C_DIS
LIN {X 0.001,Y -384.956,Z 947.792,A 0.000,B 0.000,C 90.000,E1 178.511} C_DIS
LIN {X -0.095,Y -385.512,Z 947.790,A 0.000,B 0.000,C 90.000,E1 178.165} C_DIS
LIN {X -0.168,Y -386.782,Z 947.787,A 0.000,B 0.000,C 90.000,E1 177.650} C_DIS
LIN {X 0.123,Y -389.115,Z 947.784,A 0.000,B 0.000,C 90.000,E1 177.020} C_DIS
LIN {X 0.095,Y -390.072,Z 947.783,A 0.000,B 0.000,C 90.000,E1 176.846} C_DIS
LIN {X -0.174,Y -393.821,Z 947.780,A 0.000,B 0.000,C 90.000,E1 176.331} C_DIS
LIN {X 0.138,Y -396.921,Z 947.778,A 0.000,B 0.000,C 90.000,E1 175.931} C_DIS
LIN {X -0.030,Y -399.908,Z 947.776,A 0.000,B 0.000,C 90.000,E1 175.641} C_DIS
LIN {X 0.122,Y -404.746,Z 947.773,A 0.000,B 0.000,C 90.000,E1 175.179} C_DIS
LIN {X 0.067,Y -412.439,Z 947.770,A 0.000,B 0.000,C 90.000,E1 174.546} C_DIS
LIN {X -0.207,Y -424.457,Z 947.764,A 0.000,B 0.000,C 90.000,E1 173.571} C_DIS
LIN {X 0.085,Y -432.139,Z 947.761,A 0.000,B 0.000,C 90.000,E1 172.875} C_DIS
LIN {X -0.001,Y -442.748,Z 947.755,A 0.000,B 0.000,C 90.000,E1 171.951} C_DIS
LIN {X 0.033,Y -450.081,Z 947.751,A 0.000,B 0.000,C 90.000,E1 171.254} C_DIS
LIN {X -0.008,Y -457.343,Z 947.748,A 0.000,B 0.000,C 90.000,E1 170.557} C_DIS
LIN {X -0.101,Y -464.495,Z 947.744,A 0.000,B 0.000,C 90.000,E1 169.859} C_DIS
LIN {X 0.074,Y -471.279,Z 947.740,A 0.000,B 0.000,C 90.000,E1 169.106} C_DIS
LIN {X 0.208,Y -480.547,Z 947.734,A 0.000,B 0.000,C 90.000,E1 168.049} C_DIS
LIN {X -0.192,Y -490.330,Z 947.727,A 0.000,B 0.000,C 90.000,E1 166.881} C_DIS
LIN {X -0.170,Y -496.244,Z 947.723,A 0.000,B 0.000,C 90.000,E1 166.117} C_DIS
LIN {X 0.035,Y -501.751,Z 947.719,A 0.000,B 0.000,C 90.000,E1 165.338} C_DIS
LIN {X 0.109,Y -509.053,Z 947.713,A 0.000,B 0.000,C 90.000,E1 164.283} C_DIS
LIN {X -0.045,Y -514.004,Z 947.709,A 0.000,B 0.000,C 90.000,E1 163.559} C_DIS
LIN {X 0.044,Y -520.638,Z 947.703,A 0.000,B 0.000,C 90.000,E1 162.543} C_DIS
LIN {X -0.143,Y -526.148,Z 947.698,A 0.000,B 0.000,C 90.000,E1 161.692} C_DIS
LIN {X 0.190,Y -528.906,Z 947.696,A 0.000,B 0.000,C 90.000,E1 161.221} C_DIS
LIN {X 0.116,Y -536.983,Z 947.689,A 0.000,B 0.000,C 90.000,E1 159.934} C_DIS
LIN {X -0.059,Y -545.634,Z 947.681,A 0.000,B 0.000,C 90.000,E1 158.539} C_DIS
LIN {X -0.047,Y -552.295,Z 947.674,A 0.000,B 0.000,C 90.000,E1 157.411} C_DIS
LIN {X -0.042,Y -557.808,Z 947.669,A 0.000,B 0.000,C 90.000,E1 156.433} C_DIS
LIN {X -0.064,Y -561.620,Z 947.665,A 0.000,B 0.000,C 90.000,E1 155.741} C_DIS
LIN {X 0.087,Y -568.003,Z 947.658,A 0.000,B 0.000,C 90.000,E1 154.485} C_DIS
LIN {X 0.065,Y -570.080,Z 947.656,A 0.000,B 0.000,C 90.000,E1 154.076} C_DIS
LIN {X -0.165,Y -575.743,Z 947.649,A 0.000,B 0.000,C 90.000,E1 152.871} C_DIS
LIN {X 0.091,Y -580.053,Z 947.644,A 0.000,B 0.000,C 90.000,E1 151.897} C_DIS
LIN {X -0.179,Y -584.402,Z 947.638,A 0.000,B 0.000,C 90.000,E1 150.845} C_DIS
LIN {X 0.238,Y -587.648,Z 947.633,A 0.000,B 0.000,C 90.000,E1 149.999} C_DIS
LIN {X 0.064,Y -591.674,Z 947.628,A 0.000,B 0.000,C 90.000,E1 148.948} C_DIS
LIN {X -0.360,Y -596.444,Z 947.620,A 0.000,B 0.000,C 90.000,E1 147.661} C_DIS
LIN {X 0.366,Y -601.972,Z 947.611,A 0.000,B 0.000,C 90.000,E1 146.008} C_DIS
LIN {X 0.192,Y -605.579,Z 947.606,A 0.000,B 0.000,C 90.000,E1 144.975} C_DIS
LIN {X 0.120,Y -610.985,Z 947.597,A 0.000,B 0.000,C 90.000,E1 143.417} C_DIS
LIN {X 0.227,Y -615.389,Z 947.590,A 0.000,B 0.000,C 90.000,E1 142.110} C_DIS
LIN {X -0.145,Y -620.758,Z 947.581,A 0.000,B 0.000,C 90.000,E1 140.598} C_DIS
LIN {X -0.236,Y -630.533,Z 947.565,A 0.000,B 0.000,C 90.000,E1 137.796} C_DIS
LIN {X 0.195,Y -634.351,Z 947.560,A 0.000,B 0.000,C 90.000,E1 136.743} C_DIS
LIN {X 0.065,Y -639.935,Z 947.551,A 0.000,B 0.000,C 90.000,E1 135.243} C_DIS
LIN {X -0.346,Y -644.585,Z 947.544,A 0.000,B 0.000,C 90.000,E1 134.028} C_DIS
LIN {X 0.142,Y -651.045,Z 947.535,A 0.000,B 0.000,C 90.000,E1 132.243} C_DIS
LIN {X -0.182,Y -658.462,Z 947.524,A 0.000,B 0.000,C 90.000,E1 130.297} C_DIS
LIN {X -0.211,Y -664.092,Z 947.516,A 0.000,B 0.000,C 90.000,E1 128.830} C_DIS
LIN {X -0.128,Y -669.606,Z 947.508,A 0.000,B 0.000,C 90.000,E1 127.363} C_DIS
LIN {X -0.050,Y -672.306,Z 947.504,A 0.000,B 0.000,C 90.000,E1 126.629} C_DIS
LIN {X -0.220,Y -676.495,Z 947.497,A 0.000,B 0.000,C 90.000,E1 125.438} C_DIS
LIN {X 0.070,Y -679.618,Z 947.492,A 0.000,B 0.000,C 90.000,E1 124.452} C_DIS
LIN {X 0.406,Y -681.791,Z 947.487,A 0.000,B 0.000,C 90.000,E1 123.706} C_DIS
LIN {X 0.391,Y -684.558,Z 947.482,A 0.000,B 0.000,C 90.000,E1 122.752} C_DIS
LIN {X 0.409,Y -687.041,Z 947.477,A 0.000,B 0.000,C 90.000,E1 121.799} C_DIS
LIN {X -0.268,Y -689.839,Z 947.470,A 0.000,B 0.000,C 90.000,E1 120.669} C_DIS
LIN {X 0.403,Y -691.671,Z 947.465,A 0.000,B 0.000,C 90.000,E1 119.667} C_DIS
LIN {X 0.150,Y -693.193,Z 947.460,A 0.000,B 0.000,C 90.000,E1 118.743} C_DIS
LIN {X 0.276,Y -694.182,Z 947.456,A 0.000,B 0.000,C 90.000,E1 118.025} C_DIS
LIN {X -0.277,Y -695.120,Z 947.451,A 0.000,B 0.000,C 90.000,E1 117.129} C_DIS
LIN {X 0.117,Y -695.655,Z 947.445,A 0.000,B 0.000,C 90.000,E1 116.155} C_DIS
LIN {X 0.168,Y -695.971,Z 947.439,A 0.000,B 0.000,C 90.000,E1 114.975} C_DIS
LIN {X 0.302,Y -695.930,Z 947.435,A 0.000,B 0.000,C 90.000,E1 114.259} C_DIS
LIN {X -0.111,Y -695.700,Z 947.432,A 0.000,B 0.000,C 90.000,E1 113.823} C_DIS
LIN {X 0.115,Y -694.831,Z 947.430,A 0.000,B 0.000,C 90.000,E1 113.334} C_DIS
LIN {X 0.364,Y -694.162,Z 947.428,A 0.000,B 0.000,C 90.000,E1 113.078} C_DIS
LIN {X -0.055,Y -691.655,Z 947.426,A 0.000,B 0.000,C 90.000,E1 112.642} C_DIS
LIN {X 0.063,Y -690.915,Z 947.425,A 0.000,B 0.000,C 90.000,E1 112.514} C_DIS
LIN {X 0.180,Y -689.839,Z 947.424,A 0.000,B 0.000,C 90.000,E1 112.386} C_DIS
LIN {X 0.033,Y -688.198,Z 947.424,A 0.000,B 0.000,C 90.000,E1 112.280} C_DIS
LIN {X 0.147,Y -686.050,Z 947.423,A 0.000,B 0.000,C 90.000,E1 112.153} C_DIS
LIN {X 0.396,Y -682.450,Z 947.422,A 0.000,B 0.000,C 90.000,E1 111.897} C_DIS
LIN {X -0.098,Y -680.306,Z 947.421,A 0.000,B 0.000,C 90.000,E1 111.844} C_DIS
LIN {X -0.291,Y -675.630,Z 947.421,A 0.000,B 0.000,C 90.000,E1 111.716} C_DIS
LIN {X 0.135,Y -667.369,Z 947.420,A 0.000,B 0.000,C 90.000,E1 111.589} C_DIS
LIN {X 0.099,Y -663.255,Z 947.420,A 0.000,B 0.000,C 90.000,E1 111.589} C_DIS
LIN {X 0.061,Y -634.711,Z 947.420,A 0.000,B 0.000,C 90.000,E1 111.589} C_DIS
LIN {X -0.371,Y -627.566,Z 947.419,A 0.000,B 0.000,C 90.000,E1 111.535} C_DIS
LIN {X -0.191,Y -621.756,Z 947.419,A 0.000,B 0.000,C 90.000,E1 111.408} C_DIS
LIN {X -0.309,Y -614.850,Z 947.418,A 0.000,B 0.000,C 90.000,E1 111.227} C_DIS
LIN {X -0.091,Y -608.405,Z 947.417,A 0.000,B 0.000,C 90.000,E1 110.972} C_DIS
LIN {X 0.167,Y -600.218,Z 947.414,A 0.000,B 0.000,C 90.000,E1 110.556} C_DIS
LIN {X -0.027,Y -592.936,Z 947.412,A 0.000,B 0.000,C 90.000,E1 110.120} C_DIS
LIN {X 0.263,Y -585.677,Z 947.409,A 0.000,B 0.000,C 90.000,E1 109.577} C_DIS
LIN {X -0.056,Y -576.821,Z 947.405,A 0.000,B 0.000,C 90.000,E1 108.960} C_DIS
LIN {X 0.000,Y -568.361,Z 947.403,A 0.000,B 0.000,C 90.000,E1 108.489} C_DIS
LIN {X 0.062,Y -553.992,Z 947.399,A 0.000,B 0.000,C 90.000,E1 107.819} C_DIS
LIN {X 0.205,Y -553.338,Z 947.399,A 0.000,B 0.000,C 90.000,E1 107.764} C_DIS
LIN {X -0.106,Y -551.728,Z 947.398,A 0.000,B 0.000,C 90.000,E1 107.638} C_DIS
LIN {X -0.138,Y -551.716,Z 947.398,A 0.000,B 0.000,C 90.000,E1 107.638} C_DIS
LIN {X 0.071,Y -551.232,Z 947.396,A 0.000,B 0.000,C 90.000,E1 107.347} C_DIS
LIN {X -0.222,Y -551.354,Z 947.393,A 0.000,B 0.000,C 90.000,E1 106.677} C_DIS
LIN {X -0.281,Y -551.701,Z 947.388,A 0.000,B 0.000,C 90.000,E1 105.843} C_DIS
LIN {X 0.076,Y -553.034,Z 947.372,A 0.000,B 0.000,C 90.000,E1 103.008} C_DIS
LIN {X 0.247,Y -555.119,Z 947.357,A 0.000,B 0.000,C 90.000,E1 100.197} C_DIS
LIN {X -0.160,Y -556.609,Z 947.348,A 0.000,B 0.000,C 90.000,E1 98.568} C_DIS
LIN {X -0.076,Y -558.005,Z 947.338,A 0.000,B 0.000,C 90.000,E1 96.891} C_DIS
LIN {X -0.234,Y -558.791,Z 947.332,A 0.000,B 0.000,C 90.000,E1 95.796} C_DIS
LIN {X 0.257,Y -559.665,Z 947.324,A 0.000,B 0.000,C 90.000,E1 94.359} C_DIS
LIN {X -0.268,Y -560.612,Z 947.315,A 0.000,B 0.000,C 90.000,E1 92.751} C_DIS
LIN {X 0.125,Y -561.122,Z 947.309,A 0.000,B 0.000,C 90.000,E1 91.604} C_DIS
LIN {X 0.048,Y -561.696,Z 947.301,A 0.000,B 0.000,C 90.000,E1 90.229} C_DIS
LIN {X -0.016,Y -562.141,Z 947.294,A 0.000,B 0.000,C 90.000,E1 88.854} C_DIS
LIN {X -0.062,Y -562.443,Z 947.286,A 0.000,B 0.000,C 90.000,E1 87.478} C_DIS
LIN {X -0.104,Y -562.705,Z 947.278,A 0.000,B 0.000,C 90.000,E1 86.102} C_DIS
LIN {X 0.127,Y -563.008,Z 947.268,A 0.000,B 0.000,C 90.000,E1 84.147} C_DIS
LIN {X -0.214,Y -563.297,Z 947.258,A 0.000,B 0.000,C 90.000,E1 82.527} C_DIS
LIN {X 0.014,Y -564.073,Z 947.243,A 0.000,B 0.000,C 90.000,E1 79.746} C_DIS
LIN {X -0.099,Y -564.826,Z 947.234,A 0.000,B 0.000,C 90.000,E1 78.105} C_DIS
LIN {X 0.141,Y -566.124,Z 947.222,A 0.000,B 0.000,C 90.000,E1 75.880} C_DIS
LIN {X -0.204,Y -567.112,Z 947.213,A 0.000,B 0.000,C 90.000,E1 74.267} C_DIS
LIN {X 0.028,Y -568.208,Z 947.203,A 0.000,B 0.000,C 90.000,E1 72.598} C_DIS
LIN {X 0.059,Y -569.240,Z 947.193,A 0.000,B 0.000,C 90.000,E1 70.678} C_DIS
LIN {X -0.172,Y -569.639,Z 947.188,A 0.000,B 0.000,C 90.000,E1 69.880} C_DIS
LIN {X -0.087,Y -570.188,Z 947.179,A 0.000,B 0.000,C 90.000,E1 68.230} C_DIS
LIN {X 0.039,Y -570.683,Z 947.168,A 0.000,B 0.000,C 90.000,E1 66.305} C_DIS
LIN {X 0.056,Y -571.050,Z 947.159,A 0.000,B 0.000,C 90.000,E1 64.665} C_DIS
LIN {X -0.180,Y -571.218,Z 947.150,A 0.000,B 0.000,C 90.000,E1 63.050} C_DIS
LIN {X -0.071,Y -571.397,Z 947.144,A 0.000,B 0.000,C 90.000,E1 61.948} C_DIS
LIN {X 0.311,Y -571.451,Z 947.134,A 0.000,B 0.000,C 90.000,E1 59.999} C_DIS
LIN {X -0.141,Y -571.588,Z 947.124,A 0.000,B 0.000,C 90.000,E1 58.408} C_DIS
LIN {X -0.118,Y -571.404,Z 947.117,A 0.000,B 0.000,C 90.000,E1 57.041} C_DIS
LIN {X 0.034,Y -570.889,Z 947.108,A 0.000,B 0.000,C 90.000,E1 55.388} C_DIS
LIN {X -0.097,Y -570.365,Z 947.100,A 0.000,B 0.000,C 90.000,E1 54.036} C_DIS
LIN {X 0.091,Y -569.641,Z 947.094,A 0.000,B 0.000,C 90.000,E1 52.924} C_DIS
LIN {X 0.152,Y -568.701,Z 947.088,A 0.000,B 0.000,C 90.000,E1 51.823} C_DIS
LIN {X 0.082,Y -567.891,Z 947.083,A 0.000,B 0.000,C 90.000,E1 51.009} C_DIS
LIN {X 0.121,Y -566.594,Z 947.077,A 0.000,B 0.000,C 90.000,E1 49.908} C_DIS
LIN {X 0.025,Y -565.462,Z 947.073,A 0.000,B 0.000,C 90.000,E1 49.094} C_DIS
LIN {X 0.286,Y -564.143,Z 947.068,A 0.000,B 0.000,C 90.000,E1 48.243} C_DIS
LIN {X -0.260,Y -562.562,Z 947.064,A 0.000,B 0.000,C 90.000,E1 47.472} C_DIS
LIN {X -0.113,Y -561.475,Z 947.061,A 0.000,B 0.000,C 90.000,E1 46.905} C_DIS
LIN {X 0.106,Y -559.570,Z 947.056,A 0.000,B 0.000,C 90.000,E1 46.053} C_DIS
LIN {X -0.100,Y -557.400,Z 947.051,A 0.000,B 0.000,C 90.000,E1 45.243} C_DIS
LIN {X 0.015,Y -555.834,Z 947.048,A 0.000,B 0.000,C 90.000,E1 44.676} C_DIS
LIN {X -0.229,Y -553.157,Z 947.044,A 0.000,B 0.000,C 90.000,E1 43.866} C_DIS
LIN {X -0.148,Y -551.261,Z 947.041,A 0.000,B 0.000,C 90.000,E1 43.299} C_DIS
LIN {X -0.041,Y -548.056,Z 947.036,A 0.000,B 0.000,C 90.000,E1 42.447} C_DIS
LIN {X 0.031,Y -544.508,Z 947.031,A 0.000,B 0.000,C 90.000,E1 41.595} C_DIS
LIN {X 0.255,Y -542.574,Z 947.029,A 0.000,B 0.000,C 90.000,E1 41.148} C_DIS
LIN {X 0.088,Y -537.582,Z 947.023,A 0.000,B 0.000,C 90.000,E1 40.172} C_DIS
LIN {X 0.031,Y -532.795,Z 947.018,A 0.000,B 0.000,C 90.000,E1 39.322} C_DIS
LIN {X -0.005,Y -527.740,Z 947.014,A 0.000,B 0.000,C 90.000,E1 38.463} C_DIS
LIN {X -0.089,Y -522.402,Z 947.009,A 0.000,B 0.000,C 90.000,E1 37.604} C_DIS
LIN {X 0.006,Y -519.669,Z 947.006,A 0.000,B 0.000,C 90.000,E1 37.156} C_DIS
LIN {X -0.047,Y -512.711,Z 947.001,A 0.000,B 0.000,C 90.000,E1 36.137} C_DIS
LIN {X 0.022,Y -507.460,Z 946.997,A 0.000,B 0.000,C 90.000,E1 35.391} C_DIS
LIN {X 0.024,Y -504.147,Z 946.994,A 0.000,B 0.000,C 90.000,E1 34.945} C_DIS
LIN {X 0.255,Y -498.376,Z 946.990,A 0.000,B 0.000,C 90.000,E1 34.199} C_DIS
LIN {X -0.076,Y -494.521,Z 946.988,A 0.000,B 0.000,C 90.000,E1 33.785} C_DIS
LIN {X 0.183,Y -486.499,Z 946.983,A 0.000,B 0.000,C 90.000,E1 32.880} C_DIS
LIN {X -0.141,Y -478.221,Z 946.978,A 0.000,B 0.000,C 90.000,E1 32.084} C_DIS
LIN {X -0.011,Y -472.380,Z 946.975,A 0.000,B 0.000,C 90.000,E1 31.514} C_DIS
LIN {X -0.141,Y -463.546,Z 946.971,A 0.000,B 0.000,C 90.000,E1 30.718} C_DIS
LIN {X 0.017,Y -454.709,Z 946.966,A 0.000,B 0.000,C 90.000,E1 29.922} C_DIS
LIN {X -0.153,Y -445.438,Z 946.962,A 0.000,B 0.000,C 90.000,E1 29.155} C_DIS
LIN {X -0.019,Y -427.324,Z 946.953,A 0.000,B 0.000,C 90.000,E1 27.590} C_DIS
LIN {X 0.010,Y -409.464,Z 946.944,A 0.000,B 0.000,C 90.000,E1 25.924} C_DIS
LIN {X -0.112,Y -399.289,Z 946.938,A 0.000,B 0.000,C 90.000,E1 24.899} C_DIS
LIN {X -0.072,Y -395.658,Z 946.936,A 0.000,B 0.000,C 90.000,E1 24.463} C_DIS
LIN {X -0.001,Y -393.462,Z 946.934,A 0.000,B 0.000,C 90.000,E1 24.155} C_DIS
LIN {X 0.083,Y -391.409,Z 946.932,A 0.000,B 0.000,C 90.000,E1 23.695} C_DIS
LIN {X 0.050,Y -390.841,Z 946.931,A 0.000,B 0.000,C 90.000,E1 23.590} C_DIS
LIN {X 0.010,Y -389.559,Z 946.928,A 0.000,B 0.000,C 90.000,E1 23.025} C_DIS
LIN {X -0.131,Y -389.114,Z 946.924,A 0.000,B 0.000,C 90.000,E1 22.333} C_DIS
LIN {X -0.018,Y -390.389,Z 946.913,A 0.000,B 0.000,C 90.000,E1 20.355} C_DIS
LIN {X -0.025,Y -393.196,Z 946.897,A 0.000,B 0.000,C 90.000,E1 17.511} C_DIS
LIN {X 0.105,Y -396.535,Z 946.882,A 0.000,B 0.000,C 90.000,E1 14.662} C_DIS
LIN {X -0.202,Y -399.931,Z 946.868,A 0.000,B 0.000,C 90.000,E1 12.243} C_DIS
LIN {X -0.125,Y -404.933,Z 946.850,A 0.000,B 0.000,C 90.000,E1 9.086} C_DIS
LIN {X -0.127,Y -410.534,Z 946.833,A 0.000,B 0.000,C 90.000,E1 5.967} C_DIS
LIN {X -0.026,Y -417.548,Z 946.814,A 0.000,B 0.000,C 90.000,E1 2.522} C_DIS
LIN {X -0.167,Y -425.733,Z 946.795,A 0.000,B 0.000,C 90.000,E1 359.141} C_DIS
LIN {X -0.056,Y -428.259,Z 946.791,A 0.000,B 0.000,C 90.000,E1 358.453} C_DIS
LIN {X 0.138,Y -430.327,Z 946.789,A 0.000,B 0.000,C 90.000,E1 358.051} C_DIS
LIN {X 0.172,Y -431.406,Z 946.788,A 0.000,B 0.000,C 90.000,E1 357.879} C_DIS
LIN {X -0.170,Y -435.438,Z 946.786,A 0.000,B 0.000,C 90.000,E1 357.478} C_DIS
LIN {X 0.151,Y -440.577,Z 946.784,A 0.000,B 0.000,C 90.000,E1 357.078} C_DIS
LIN {X 0.148,Y -458.904,Z 946.779,A 0.000,B 0.000,C 90.000,E1 356.159} C_DIS
LIN {X -0.076,Y -467.192,Z 946.776,A 0.000,B 0.000,C 90.000,E1 355.755} C_DIS
LIN {X -0.093,Y -482.456,Z 946.772,A 0.000,B 0.000,C 90.000,E1 354.951} C_DIS
LIN {X 0.008,Y -497.081,Z 946.768,A 0.000,B 0.000,C 90.000,E1 354.147} C_DIS
LIN {X -0.092,Y -505.283,Z 946.765,A 0.000,B 0.000,C 90.000,E1 353.685} C_DIS
LIN {X 0.169,Y -517.969,Z 946.761,A 0.000,B 0.000,C 90.000,E1 352.875} C_DIS
LIN {X 0.150,Y -525.710,Z 946.758,A 0.000,B 0.000,C 90.000,E1 352.356} C_DIS
LIN {X -0.166,Y -533.217,Z 946.755,A 0.000,B 0.000,C 90.000,E1 351.837} C_DIS
LIN {X -0.117,Y -540.418,Z 946.751,A 0.000,B 0.000,C 90.000,E1 351.254} C_DIS
LIN {X 0.031,Y -547.366,Z 946.748,A 0.000,B 0.000,C 90.000,E1 350.622} C_DIS
LIN {X -0.106,Y -553.848,Z 946.744,A 0.000,B 0.000,C 90.000,E1 349.982} C_DIS
LIN {X -0.201,Y -558.829,Z 946.741,A 0.000,B 0.000,C 90.000,E1 349.454} C_DIS
LIN {X -0.134,Y -564.636,Z 946.737,A 0.000,B 0.000,C 90.000,E1 348.757} C_DIS
LIN {X -0.176,Y -568.794,Z 946.735,A 0.000,B 0.000,C 90.000,E1 348.229} C_DIS
LIN {X -0.177,Y -574.785,Z 946.730,A 0.000,B 0.000,C 90.000,E1 347.409} C_DIS
LIN {X 0.123,Y -579.403,Z 946.726,A 0.000,B 0.000,C 90.000,E1 346.700} C_DIS
LIN {X -0.099,Y -586.046,Z 946.720,A 0.000,B 0.000,C 90.000,E1 345.644} C_DIS
LIN {X -0.090,Y -592.116,Z 946.714,A 0.000,B 0.000,C 90.000,E1 344.574} C_DIS
LIN {X 0.300,Y -596.323,Z 946.710,A 0.000,B 0.000,C 90.000,E1 343.740} C_DIS
LIN {X -0.068,Y -600.934,Z 946.705,A 0.000,B 0.000,C 90.000,E1 342.851} C_DIS
LIN {X -0.255,Y -605.870,Z 946.699,A 0.000,B 0.000,C 90.000,E1 341.819} C_DIS
LIN {X -0.301,Y -609.495,Z 946.695,A 0.000,B 0.000,C 90.000,E1 341.040} C_DIS
LIN {X -0.378,Y -613.991,Z 946.689,A 0.000,B 0.000,C 90.000,E1 340.007} C_DIS
LIN {X -0.176,Y -618.234,Z 946.683,A 0.000,B 0.000,C 90.000,E1 338.954} C_DIS
LIN {X -0.139,Y -622.201,Z 946.677,A 0.000,B 0.000,C 90.000,E1 337.922} C_DIS
LIN {X 0.179,Y -625.985,Z 946.672,A 0.000,B 0.000,C 90.000,E1 336.869} C_DIS
LIN {X -0.008,Y -630.234,Z 946.665,A 0.000,B 0.000,C 90.000,E1 335.613} C_DIS
LIN {X 0.146,Y -634.156,Z 946.658,A 0.000,B 0.000,C 90.000,E1 334.332} C_DIS
LIN {X 0.088,Y -637.891,Z 946.651,A 0.000,B 0.000,C 90.000,E1 333.076} C_DIS
LIN {X -0.260,Y -640.579,Z 946.645,A 0.000,B 0.000,C 90.000,E1 332.103} C_DIS
LIN {X 0.299,Y -643.003,Z 946.639,A 0.000,B 0.000,C 90.000,E1 331.051} C_DIS
LIN {X 0.088,Y -645.834,Z 946.632,A 0.000,B 0.000,C 90.000,E1 329.822} C_DIS
LIN {X 0.018,Y -648.396,Z 946.626,A 0.000,B 0.000,C 90.000,E1 328.584} C_DIS
LIN {X 0.211,Y -650.536,Z 946.619,A 0.000,B 0.000,C 90.000,E1 327.327} C_DIS
LIN {X 0.232,Y -652.389,Z 946.612,A 0.000,B 0.000,C 90.000,E1 326.087} C_DIS
LIN {X -0.253,Y -654.019,Z 946.605,A 0.000,B 0.000,C 90.000,E1 324.895} C_DIS
LIN {X -0.256,Y -655.481,Z 946.597,A 0.000,B 0.000,C 90.000,E1 323.417} C_DIS
LIN {X -0.305,Y -656.543,Z 946.590,A 0.000,B 0.000,C 90.000,E1 322.190} C_DIS
LIN {X 0.073,Y -657.463,Z 946.583,A 0.000,B 0.000,C 90.000,E1 320.928} C_DIS
LIN {X 0.045,Y -658.424,Z 946.576,A 0.000,B 0.000,C 90.000,E1 319.703} C_DIS
LIN {X -0.084,Y -659.362,Z 946.568,A 0.000,B 0.000,C 90.000,E1 318.243} C_DIS
LIN {X -0.273,Y -661.308,Z 946.554,A 0.000,B 0.000,C 90.000,E1 315.810} C_DIS
LIN {X -0.391,Y -662.870,Z 946.544,A 0.000,B 0.000,C 90.000,E1 313.866} C_DIS
LIN {X 0.032,Y -664.019,Z 946.537,A 0.000,B 0.000,C 90.000,E1 312.609} C_DIS
LIN {X 0.020,Y -665.383,Z 946.529,A 0.000,B 0.000,C 90.000,E1 311.148} C_DIS
LIN {X 0.038,Y -666.475,Z 946.522,A 0.000,B 0.000,C 90.000,E1 309.930} C_DIS
LIN {X 0.149,Y -667.642,Z 946.514,A 0.000,B 0.000,C 90.000,E1 308.463} C_DIS
LIN {X -0.214,Y -668.318,Z 946.508,A 0.000,B 0.000,C 90.000,E1 307.523} C_DIS
LIN {X -0.053,Y -668.863,Z 946.502,A 0.000,B 0.000,C 90.000,E1 306.297} C_DIS
LIN {X -0.185,Y -669.381,Z 946.492,A 0.000,B 0.000,C 90.000,E1 304.612} C_DIS
LIN {X 0.243,Y -670.041,Z 946.483,A 0.000,B 0.000,C 90.000,E1 302.880} C_DIS
LIN {X -0.191,Y -670.772,Z 946.475,A 0.000,B 0.000,C 90.000,E1 301.465} C_DIS
LIN {X -0.072,Y -674.376,Z 946.453,A 0.000,B 0.000,C 90.000,E1 297.590} C_DIS
LIN {X 0.090,Y -677.907,Z 946.441,A 0.000,B 0.000,C 90.000,E1 295.412} C_DIS
LIN {X 0.161,Y -679.906,Z 946.435,A 0.000,B 0.000,C 90.000,E1 294.207} C_DIS
LIN {X 0.053,Y -681.358,Z 946.429,A 0.000,B 0.000,C 90.000,E1 293.259} C_DIS
LIN {X 0.383,Y -681.946,Z 946.425,A 0.000,B 0.000,C 90.000,E1 292.514} C_DIS
LIN {X -0.111,Y -681.717,Z 946.423,A 0.000,B 0.000,C 90.000,E1 292.078} C_DIS
LIN {X -0.168,Y -681.278,Z 946.421,A 0.000,B 0.000,C 90.000,E1 291.844} C_DIS
LIN {X -0.029,Y -679.135,Z 946.419,A 0.000,B 0.000,C 90.000,E1 291.354} C_DIS
LIN {X 0.066,Y -678.497,Z 946.418,A 0.000,B 0.000,C 90.000,E1 291.227} C_DIS
LIN {X 0.160,Y -677.663,Z 946.417,A 0.000,B 0.000,C 90.000,E1 291.099} C_DIS
LIN {X 0.249,Y -676.425,Z 946.417,A 0.000,B 0.000,C 90.000,E1 290.972} C_DIS
LIN {X -0.038,Y -670.840,Z 946.414,A 0.000,B 0.000,C 90.000,E1 290.556} C_DIS
LIN {X -0.073,Y -664.682,Z 946.412,A 0.000,B 0.000,C 90.000,E1 290.174} C_DIS
LIN {X -0.182,Y -661.332,Z 946.411,A 0.000,B 0.000,C 90.000,E1 289.939} C_DIS
LIN {X -0.247,Y -661.282,Z 946.411,A 0.000,B 0.000,C 90.000,E1 289.939} C_DIS
LIN {X -0.228,Y -660.589,Z 946.410,A 0.000,B 0.000,C 90.000,E1 289.812} C_DIS
LIN {X -0.273,Y -660.569,Z 946.410,A 0.000,B 0.000,C 90.000,E1 289.812} C_DIS
LIN {X 0.064,Y -660.678,Z 946.409,A 0.000,B 0.000,C 90.000,E1 289.523} C_DIS
LIN {X -0.153,Y -661.882,Z 946.406,A 0.000,B 0.000,C 90.000,E1 289.141} C_DIS
LIN {X -0.316,Y -662.364,Z 946.406,A 0.000,B 0.000,C 90.000,E1 289.033} C_DIS
LIN {X -0.309,Y -669.811,Z 946.398,A 0.000,B 0.000,C 90.000,E1 287.638} C_DIS
LIN {X 0.385,Y -672.288,Z 946.395,A 0.000,B 0.000,C 90.000,E1 287.094} C_DIS
LIN {X 0.196,Y -675.399,Z 946.391,A 0.000,B 0.000,C 90.000,E1 286.386} C_DIS
LIN {X 0.275,Y -677.159,Z 946.388,A 0.000,B 0.000,C 90.000,E1 285.898} C_DIS
LIN {X 0.135,Y -679.328,Z 946.385,A 0.000,B 0.000,C 90.000,E1 285.190} C_DIS
LIN {X 0.019,Y -681.010,Z 946.380,A 0.000,B 0.000,C 90.000,E1 284.481} C_DIS
LIN {X -0.110,Y -682.811,Z 946.375,A 0.000,B 0.000,C 90.000,E1 283.536} C_DIS
LIN {X -0.194,Y -683.887,Z 946.371,A 0.000,B 0.000,C 90.000,E1 282.827} C_DIS
LIN {X 0.374,Y -684.908,Z 946.366,A 0.000,B 0.000,C 90.000,E1 281.827} C_DIS
LIN {X 0.188,Y -685.168,Z 946.363,A 0.000,B 0.000,C 90.000,E1 281.366} C_DIS
LIN {X 0.116,Y -685.079,Z 946.359,A 0.000,B 0.000,C 90.000,E1 280.658} C_DIS
LIN {X -0.060,Y -684.657,Z 946.357,A 0.000,B 0.000,C 90.000,E1 280.197} C_DIS
LIN {X -0.118,Y -683.812,Z 946.354,A 0.000,B 0.000,C 90.000,E1 279.726} C_DIS
LIN {X -0.297,Y -682.686,Z 946.351,A 0.000,B 0.000,C 90.000,E1 279.265} C_DIS
LIN {X 0.340,Y -682.038,Z 946.350,A 0.000,B 0.000,C 90.000,E1 278.973} C_DIS
LIN {X 0.152,Y -680.383,Z 946.347,A 0.000,B 0.000,C 90.000,E1 278.511} C_DIS
LIN {X -0.041,Y -678.361,Z 946.345,A 0.000,B 0.000,C 90.000,E1 278.049} C_DIS
LIN {X -0.308,Y -674.916,Z 946.341,A 0.000,B 0.000,C 90.000,E1 277.352} C_DIS
LIN {X 0.135,Y -672.460,Z 946.338,A 0.000,B 0.000,C 90.000,E1 276.834} C_DIS
LIN {X -0.194,Y -668.977,Z 946.335,A 0.000,B 0.000,C 90.000,E1 276.258} C_DIS
LIN {X 0.204,Y -665.941,Z 946.332,A 0.000,B 0.000,C 90.000,E1 275.739} C_DIS
LIN {X -0.083,Y -662.444,Z 946.329,A 0.000,B 0.000,C 90.000,E1 275.277} C_DIS
LIN {X 0.264,Y -658.634,Z 946.327,A 0.000,B 0.000,C 90.000,E1 274.759} C_DIS
LIN {X -0.220,Y -653.152,Z 946.323,A 0.000,B 0.000,C 90.000,E1 274.188} C_DIS
LIN {X 0.062,Y -648.510,Z 946.320,A 0.000,B 0.000,C 90.000,E1 273.669} C_DIS
LIN {X -0.207,Y -642.365,Z 946.317,A 0.000,B 0.000,C 90.000,E1 273.094} C_DIS
LIN {X 0.295,Y -637.101,Z 946.315,A 0.000,B 0.000,C 90.000,E1 272.579} C_DIS
LIN {X -0.292,Y -631.628,Z 946.312,A 0.000,B 0.000,C 90.000,E1 272.178} C_DIS
LIN {X 0.115,Y -624.278,Z 946.309,A 0.000,B 0.000,C 90.000,E1 271.604} C_DIS
LIN {X -0.273,Y -616.670,Z 946.306,A 0.000,B 0.000,C 90.000,E1 271.146} C_DIS
LIN {X -0.075,Y -610.374,Z 946.304,A 0.000,B 0.000,C 90.000,E1 270.745} C_DIS
LIN {X -0.203,Y -603.802,Z 946.302,A 0.000,B 0.000,C 90.000,E1 270.401} C_DIS
LIN {X -0.051,Y -597.066,Z 946.300,A 0.000,B 0.000,C 90.000,E1 270.057} C_DIS
LIN {X -0.136,Y -590.018,Z 946.299,A 0.000,B 0.000,C 90.000,E1 269.771} C_DIS
LIN {X 0.151,Y -584.685,Z 946.298,A 0.000,B 0.000,C 90.000,E1 269.542} C_DIS
LIN {X 0.036,Y -578.615,Z 946.297,A 0.000,B 0.000,C 90.000,E1 269.370} C_DIS
LIN {X -0.160,Y -570.915,Z 946.296,A 0.000,B 0.000,C 90.000,E1 269.198} C_DIS
LIN {X -0.182,Y -564.983,Z 946.295,A 0.000,B 0.000,C 90.000,E1 269.083} C_DIS
LIN {X 0.032,Y -556.749,Z 946.294,A 0.000,B 0.000,C 90.000,E1 268.969} C_DIS
LIN {X -0.180,Y -552.162,Z 946.294,A 0.000,B 0.000,C 90.000,E1 268.969} C_DIS
LIN {X -0.166,Y -547.769,Z 946.294,A 0.000,B 0.000,C 90.000,E1 268.912} C_DIS
LIN {X 0.021,Y -544.056,Z 946.293,A 0.000,B 0.000,C 90.000,E1 268.682} C_DIS
LIN {X -0.034,Y -543.981,Z 946.293,A 0.000,B 0.000,C 90.000,E1 268.682} C_DIS
LIN {X 0.066,Y -543.562,Z 946.292,A 0.000,B 0.000,C 90.000,E1 268.511} C_DIS
LIN {X 0.097,Y -543.243,Z 946.290,A 0.000,B 0.000,C 90.000,E1 268.224} C_DIS
LIN {X 0.283,Y -541.930,Z 946.282,A 0.000,B 0.000,C 90.000,E1 266.788} C_DIS
LIN {X -0.051,Y -540.383,Z 946.271,A 0.000,B 0.000,C 90.000,E1 264.837} C_DIS
LIN {X 0.085,Y -539.619,Z 946.265,A 0.000,B 0.000,C 90.000,E1 263.685} C_DIS
LIN {X -0.203,Y -538.436,Z 946.256,A 0.000,B 0.000,C 90.000,E1 262.008} C_DIS
LIN {X -0.089,Y -537.792,Z 946.251,A 0.000,B 0.000,C 90.000,E1 261.141} C_DIS
LIN {X 0.012,Y -536.876,Z 946.246,A 0.000,B 0.000,C 90.000,E1 260.274} C_DIS
LIN {X 0.250,Y -535.380,Z 946.240,A 0.000,B 0.000,C 90.000,E1 259.106} C_DIS
LIN {X 0.094,Y -532.730,Z 946.229,A 0.000,B 0.000,C 90.000,E1 257.117} C_DIS
LIN {X 0.119,Y -530.384,Z 946.217,A 0.000,B 0.000,C 90.000,E1 255.102} C_DIS
LIN {X 0.065,Y -528.383,Z 946.208,A 0.000,B 0.000,C 90.000,E1 253.378} C_DIS
LIN {X -0.065,Y -527.076,Z 946.201,A 0.000,B 0.000,C 90.000,E1 252.236} C_DIS
LIN {X -0.055,Y -524.817,Z 946.192,A 0.000,B 0.000,C 90.000,E1 250.496} C_DIS
LIN {X 0.089,Y -522.971,Z 946.184,A 0.000,B 0.000,C 90.000,E1 249.028} C_DIS
LIN {X -0.090,Y -521.111,Z 946.175,A 0.000,B 0.000,C 90.000,E1 247.592} C_DIS
LIN {X 0.184,Y -518.998,Z 946.167,A 0.000,B 0.000,C 90.000,E1 246.102} C_DIS
LIN {X -0.065,Y -516.662,Z 946.159,A 0.000,B 0.000,C 90.000,E1 244.665} C_DIS
LIN {X -0.262,Y -514.810,Z 946.153,A 0.000,B 0.000,C 90.000,E1 243.512} C_DIS
LIN {X -0.037,Y -511.989,Z 946.143,A 0.000,B 0.000,C 90.000,E1 241.719} C_DIS
LIN {X -0.172,Y -509.592,Z 946.135,A 0.000,B 0.000,C 90.000,E1 240.255} C_DIS
LIN {X -0.017,Y -506.297,Z 946.125,A 0.000,B 0.000,C 90.000,E1 238.456} C_DIS
LIN {X 0.321,Y -502.407,Z 946.115,A 0.000,B 0.000,C 90.000,E1 236.628} C_DIS
LIN {X -0.021,Y -499.680,Z 946.108,A 0.000,B 0.000,C 90.000,E1 235.468} C_DIS
LIN {X -0.107,Y -493.581,Z 946.093,A 0.000,B 0.000,C 90.000,E1 232.763} C_DIS
LIN {X -0.003,Y -489.489,Z 946.083,A 0.000,B 0.000,C 90.000,E1 230.928} C_DIS
LIN {X 0.032,Y -486.729,Z 946.076,A 0.000,B 0.000,C 90.000,E1 229.703} C_DIS
LIN {X 0.098,Y -483.184,Z 946.068,A 0.000,B 0.000,C 90.000,E1 228.162} C_DIS
LIN {X -0.335,Y -478.366,Z 946.056,A 0.000,B 0.000,C 90.000,E1 226.053} C_DIS
LIN {X 0.235,Y -474.863,Z 946.047,A 0.000,B 0.000,C 90.000,E1 224.433} C_DIS
LIN {X -0.034,Y -472.145,Z 946.040,A 0.000,B 0.000,C 90.000,E1 223.218} C_DIS
LIN {X -0.240,Y -468.741,Z 946.031,A 0.000,B 0.000,C 90.000,E1 221.676} C_DIS
LIN {X -0.099,Y -464.512,Z 946.021,A 0.000,B 0.000,C 90.000,E1 219.769} C_DIS
LIN {X 0.216,Y -461.817,Z 946.014,A 0.000,B 0.000,C 90.000,E1 218.463} C_DIS
LIN {X 0.231,Y -458.350,Z 946.005,A 0.000,B 0.000,C 90.000,E1 216.870} C_DIS
LIN {X 0.179,Y -455.531,Z 945.998,A 0.000,B 0.000,C 90.000,E1 215.598} C_DIS
LIN {X -0.025,Y -450.576,Z 945.985,A 0.000,B 0.000,C 90.000,E1 213.372} C_DIS
LIN {X -0.167,Y -444.860,Z 945.971,A 0.000,B 0.000,C 90.000,E1 210.797} C_DIS
LIN {X 0.000,Y -439.924,Z 945.958,A 0.000,B 0.000,C 90.000,E1 208.487} C_DIS
LIN {X 0.178,Y -435.601,Z 945.947,A 0.000,B 0.000,C 90.000,E1 206.488} C_DIS
LIN {X 0.061,Y -431.915,Z 945.938,A 0.000,B 0.000,C 90.000,E1 204.847} C_DIS
LIN {X -0.125,Y -428.264,Z 945.929,A 0.000,B 0.000,C 90.000,E1 203.206} C_DIS
LIN {X -0.161,Y -424.425,Z 945.920,A 0.000,B 0.000,C 90.000,E1 201.535} C_DIS
LIN {X -0.103,Y -420.127,Z 945.908,A 0.000,B 0.000,C 90.000,E1 199.504} C_DIS
LIN {X 0.116,Y -415.261,Z 945.895,A 0.000,B 0.000,C 90.000,E1 197.094} C_DIS
LIN {X -0.190,Y -411.816,Z 945.886,A 0.000,B 0.000,C 90.000,E1 195.426} C_DIS
LIN {X 0.111,Y -409.078,Z 945.878,A 0.000,B 0.000,C 90.000,E1 194.008} C_DIS
LIN {X -0.011,Y -404.902,Z 945.866,A 0.000,B 0.000,C 90.000,E1 191.951} C_DIS
LIN {X 0.079,Y -400.935,Z 945.855,A 0.000,B 0.000,C 90.000,E1 189.849} C_DIS
LIN {X -0.002,Y -396.888,Z 945.843,A 0.000,B 0.000,C 90.000,E1 187.757} C_DIS
LIN {X 0.186,Y -393.564,Z 945.833,A 0.000,B 0.000,C 90.000,E1 185.967} C_DIS
LIN {X -0.162,Y -390.330,Z 945.823,A 0.000,B 0.000,C 90.000,E1 184.245} C_DIS
LIN {X 0.031,Y -386.173,Z 945.810,A 0.000,B 0.000,C 90.000,E1 181.718} C_DIS
LIN {X 0.113,Y -384.817,Z 945.804,A 0.000,B 0.000,C 90.000,E1 180.630} C_DIS
LIN {X -0.096,Y -384.256,Z 945.800,A 0.000,B 0.000,C 90.000,E1 179.943} C_DIS
LIN {X 0.016,Y -384.009,Z 945.794,A 0.000,B 0.000,C 90.000,E1 178.854} C_DIS
LIN {X -0.093,Y -384.157,Z 945.792,A 0.000,B 0.000,C 90.000,E1 178.511} C_DIS
LIN {X 0.165,Y -385.153,Z 945.788,A 0.000,B 0.000,C 90.000,E1 177.764} C_DIS
LIN {X 0.003,Y -386.557,Z 945.785,A 0.000,B 0.000,C 90.000,E1 177.249} C_DIS
LIN {X -0.133,Y -388.690,Z 945.782,A 0.000,B 0.000,C 90.000,E1 176.731} C_DIS
LIN {X 0.067,Y -393.322,Z 945.778,A 0.000,B 0.000,C 90.000,E1 175.988} C_DIS
LIN {X 0.062,Y -395.873,Z 945.776,A 0.000,B 0.000,C 90.000,E1 175.698} C_DIS
LIN {X 0.005,Y -400.421,Z 945.774,A 0.000,B 0.000,C 90.000,E1 175.241} C_DIS
LIN {X -0.072,Y -411.412,Z 945.768,A 0.000,B 0.000,C 90.000,E1 174.318} C_DIS
LIN {X 0.192,Y -425.652,Z 945.762,A 0.000,B 0.000,C 90.000,E1 173.109} C_DIS
LIN {X -0.224,Y -436.332,Z 945.757,A 0.000,B 0.000,C 90.000,E1 172.243} C_DIS
LIN {X -0.174,Y -440.951,Z 945.755,A 0.000,B 0.000,C 90.000,E1 171.837} C_DIS
LIN {X -0.019,Y -451.223,Z 945.749,A 0.000,B 0.000,C 90.000,E1 170.849} C_DIS
LIN {X 0.204,Y -459.945,Z 945.745,A 0.000,B 0.000,C 90.000,E1 169.982} C_DIS
LIN {X -0.134,Y -465.541,Z 945.741,A 0.000,B 0.000,C 90.000,E1 169.454} C_DIS
LIN {X -0.158,Y -471.026,Z 945.738,A 0.000,B 0.000,C 90.000,E1 168.870} C_DIS
LIN {X 0.139,Y -479.179,Z 945.733,A 0.000,B 0.000,C 90.000,E1 167.937} C_DIS
LIN {X -0.079,Y -490.245,Z 945.725,A 0.000,B 0.000,C 90.000,E1 166.589} C_DIS
LIN {X -0.058,Y -496.177,Z 945.721,A 0.000,B 0.000,C 90.000,E1 165.825} C_DIS
LIN {X 0.148,Y -501.609,Z 945.717,A 0.000,B 0.000,C 90.000,E1 165.046} C_DIS
LIN {X -0.211,Y -506.974,Z 945.713,A 0.000,B 0.000,C 90.000,E1 164.338} C_DIS
LIN {X 0.106,Y -511.908,Z 945.709,A 0.000,B 0.000,C 90.000,E1 163.559} C_DIS
LIN {X 0.011,Y -518.817,Z 945.703,A 0.000,B 0.000,C 90.000,E1 162.543} C_DIS
LIN {X -0.009,Y -523.341,Z 945.699,A 0.000,B 0.000,C 90.000,E1 161.819} C_DIS
LIN {X -0.152,Y -526.269,Z 945.697,A 0.000,B 0.000,C 90.000,E1 161.402} C_DIS
LIN {X 0.076,Y -535.221,Z 945.689,A 0.000,B 0.000,C 90.000,E1 159.934} C_DIS
LIN {X 0.165,Y -539.541,Z 945.685,A 0.000,B 0.000,C 90.000,E1 159.209} C_DIS
LIN {X -0.221,Y -544.022,Z 945.681,A 0.000,B 0.000,C 90.000,E1 158.539} C_DIS
LIN {X 0.153,Y -551.565,Z 945.674,A 0.000,B 0.000,C 90.000,E1 157.230} C_DIS
LIN {X 0.262,Y -557.856,Z 945.667,A 0.000,B 0.000,C 90.000,E1 156.102} C_DIS
LIN {X 0.248,Y -561.630,Z 945.664,A 0.000,B 0.000,C 90.000,E1 155.409} C_DIS
LIN {X -0.194,Y -568.722,Z 945.656,A 0.000,B 0.000,C 90.000,E1 154.076} C_DIS
LIN {X 0.065,Y -574.517,Z 945.649,A 0.000,B 0.000,C 90.000,E1 152.820} C_DIS
LIN {X -0.209,Y -578.820,Z 945.644,A 0.000,B 0.000,C 90.000,E1 151.897} C_DIS
LIN {X 0.012,Y -583.333,Z 945.638,A 0.000,B 0.000,C 90.000,E1 150.795} C_DIS
LIN {X -0.094,Y -586.597,Z 945.633,A 0.000,B 0.000,C 90.000,E1 149.999} C_DIS
LIN {X 0.021,Y -590.698,Z 945.627,A 0.000,B 0.000,C 90.000,E1 148.918} C_DIS
LIN {X 0.095,Y -595.528,Z 945.620,A 0.000,B 0.000,C 90.000,E1 147.582} C_DIS
LIN {X -0.263,Y -600.220,Z 945.613,A 0.000,B 0.000,C 90.000,E1 146.294} C_DIS
LIN {X 0.124,Y -603.044,Z 945.608,A 0.000,B 0.000,C 90.000,E1 145.468} C_DIS
LIN {X 0.272,Y -609.360,Z 945.598,A 0.000,B 0.000,C 90.000,E1 143.623} C_DIS
LIN {X -0.211,Y -614.698,Z 945.589,A 0.000,B 0.000,C 90.000,E1 142.110} C_DIS
LIN {X 0.271,Y -620.104,Z 945.581,A 0.000,B 0.000,C 90.000,E1 140.517} C_DIS
LIN {X 0.044,Y -624.457,Z 945.574,A 0.000,B 0.000,C 90.000,E1 139.256} C_DIS
LIN {X -0.189,Y -632.930,Z 945.561,A 0.000,B 0.000,C 90.000,E1 136.986} C_DIS
LIN {X -0.351,Y -638.582,Z 945.553,A 0.000,B 0.000,C 90.000,E1 135.486} C_DIS
LIN {X 0.046,Y -644.188,Z 945.544,A 0.000,B 0.000,C 90.000,E1 133.947} C_DIS
LIN {X 0.045,Y -650.697,Z 945.535,A 0.000,B 0.000,C 90.000,E1 132.204} C_DIS
LIN {X 0.239,Y -657.228,Z 945.525,A 0.000,B 0.000,C 90.000,E1 130.458} C_DIS
LIN {X 0.193,Y -662.861,Z 945.517,A 0.000,B 0.000,C 90.000,E1 128.991} C_DIS
LIN {X -0.244,Y -667.457,Z 945.510,A 0.000,B 0.000,C 90.000,E1 127.810} C_DIS
LIN {X 0.332,Y -671.171,Z 945.505,A 0.000,B 0.000,C 90.000,E1 126.790} C_DIS
LIN {X -0.253,Y -676.202,Z 945.497,A 0.000,B 0.000,C 90.000,E1 125.391} C_DIS
LIN {X -0.123,Y -678.605,Z 945.493,A 0.000,B 0.000,C 90.000,E1 124.659} C_DIS
LIN {X 0.202,Y -680.845,Z 945.489,A 0.000,B 0.000,C 90.000,E1 123.913} C_DIS
LIN {X -0.209,Y -684.328,Z 945.482,A 0.000,B 0.000,C 90.000,E1 122.752} C_DIS
LIN {X 0.181,Y -686.237,Z 945.478,A 0.000,B 0.000,C 90.000,E1 122.005} C_DIS
LIN {X -0.156,Y -689.006,Z 945.471,A 0.000,B 0.000,C 90.000,E1 120.846} C_DIS
LIN {X 0.292,Y -690.019,Z 945.469,A 0.000,B 0.000,C 90.000,E1 120.335} C_DIS
LIN {X -0.213,Y -691.355,Z 945.465,A 0.000,B 0.000,C 90.000,E1 119.667} C_DIS
LIN {X 0.137,Y -692.876,Z 945.460,A 0.000,B 0.000,C 90.000,E1 118.693} C_DIS
LIN {X 0.263,Y -693.834,Z 945.456,A 0.000,B 0.000,C 90.000,E1 117.975} C_DIS
LIN {X 0.028,Y -694.770,Z 945.450,A 0.000,B 0.000,C 90.000,E1 117.052} C_DIS
LIN {X 0.105,Y -695.257,Z 945.445,A 0.000,B 0.000,C 90.000,E1 116.104} C_DIS
LIN {X -0.181,Y -695.532,Z 945.439,A 0.000,B 0.000,C 90.000,E1 114.951} C_DIS
LIN {X 0.035,Y -695.554,Z 945.436,A 0.000,B 0.000,C 90.000,E1 114.463} C_DIS
LIN {X -0.093,Y -695.334,Z 945.433,A 0.000,B 0.000,C 90.000,E1 114.003} C_DIS
LIN {X -0.123,Y -695.126,Z 945.432,A 0.000,B 0.000,C 90.000,E1 113.770} C_DIS
LIN {X 0.375,Y -694.293,Z 945.429,A 0.000,B 0.000,C 90.000,E1 113.259} C_DIS
LIN {X -0.289,Y -693.417,Z 945.428,A 0.000,B 0.000,C 90.000,E1 113.078} C_DIS
LIN {X -0.071,Y -690.993,Z 945.426,A 0.000,B 0.000,C 90.000,E1 112.589} C_DIS
LIN {X 0.047,Y -690.095,Z 945.425,A 0.000,B 0.000,C 90.000,E1 112.461} C_DIS
LIN {X 0.164,Y -688.755,Z 945.424,A 0.000,B 0.000,C 90.000,E1 112.333} C_DIS
LIN {X -0.176,Y -682.437,Z 945.422,A 0.000,B 0.000,C 90.000,E1 111.950} C_DIS
LIN {X -0.038,Y -680.332,Z 945.421,A 0.000,B 0.000,C 90.000,E1 111.844} C_DIS
LIN {X 0.353,Y -677.562,Z 945.421,A 0.000,B 0.000,C 90.000,E1 111.716} C_DIS
LIN {X -0.274,Y -675.622,Z 945.421,A 0.000,B 0.000,C 90.000,E1 111.716} C_DIS
LIN {X 0.093,Y -667.923,Z 945.420,A 0.000,B 0.000,C 90.000,E1 111.589} C_DIS
LIN {X -0.076,Y -660.718,Z 945.420,A 0.000,B 0.000,C 90.000,E1 111.589} C_DIS
LIN {X -0.134,Y -634.992,Z 945.420,A 0.000,B 0.000,C 90.000,E1 111.589} C_DIS
LIN {X -0.279,Y -629.474,Z 945.420,A 0.000,B 0.000,C 90.000,E1 111.535} C_DIS
LIN {X -0.317,Y -622.287,Z 945.419,A 0.000,B 0.000,C 90.000,E1 111.408} C_DIS
LIN {X 0.154,Y -615.217,Z 945.418,A 0.000,B 0.000,C 90.000,E1 111.173} C_DIS
LIN {X 0.141,Y -608.227,Z 945.416,A 0.000,B 0.000,C 90.000,E1 110.918} C_DIS
LIN {X -0.196,Y -600.047,Z 945.414,A 0.000,B 0.000,C 90.000,E1 110.556} C_DIS
LIN {X -0.141,Y -593.131,Z 945.412,A 0.000,B 0.000,C 90.000,E1 110.120} C_DIS
LIN {X -0.118,Y -576.995,Z 945.405,A 0.000,B 0.000,C 90.000,E1 108.960} C_DIS
LIN {X -0.059,Y -568.527,Z 945.403,A 0.000,B 0.000,C 90.000,E1 108.489} C_DIS
LIN {X -0.291,Y -553.514,Z 945.399,A 0.000,B 0.000,C 90.000,E1 107.819} C_DIS
LIN {X -0.029,Y -551.871,Z 945.398,A 0.000,B 0.000,C 90.000,E1 107.638} C_DIS
LIN {X -0.067,Y -551.848,Z 945.398,A 0.000,B 0.000,C 90.000,E1 107.638} C_DIS
LIN {X 0.018,Y -551.483,Z 945.397,A 0.000,B 0.000,C 90.000,E1 107.457} C_DIS
LIN {X 0.120,Y -551.368,Z 945.396,A 0.000,B 0.000,C 90.000,E1 107.166} C_DIS
LIN {X -0.096,Y -551.860,Z 945.388,A 0.000,B 0.000,C 90.000,E1 105.788} C_DIS
LIN {X -0.266,Y -553.184,Z 945.372,A 0.000,B 0.000,C 90.000,E1 103.008} C_DIS
LIN {X -0.090,Y -555.263,Z 945.357,A 0.000,B 0.000,C 90.000,E1 100.197} C_DIS
LIN {X 0.055,Y -556.742,Z 945.347,A 0.000,B 0.000,C 90.000,E1 98.511} C_DIS
LIN {X 0.144,Y -558.109,Z 945.338,A 0.000,B 0.000,C 90.000,E1 96.834} C_DIS
LIN {X -0.011,Y -558.886,Z 945.332,A 0.000,B 0.000,C 90.000,E1 95.739} C_DIS
LIN {X -0.074,Y -559.746,Z 945.324,A 0.000,B 0.000,C 90.000,E1 94.359} C_DIS
LIN {X -0.038,Y -560.695,Z 945.315,A 0.000,B 0.000,C 90.000,E1 92.694} C_DIS
LIN {X -0.204,Y -561.197,Z 945.309,A 0.000,B 0.000,C 90.000,E1 91.604} C_DIS
LIN {X -0.280,Y -561.758,Z 945.301,A 0.000,B 0.000,C 90.000,E1 90.229} C_DIS
LIN {X 0.217,Y -562.192,Z 945.294,A 0.000,B 0.000,C 90.000,E1 88.797} C_DIS
LIN {X 0.173,Y -562.511,Z 945.286,A 0.000,B 0.000,C 90.000,E1 87.421} C_DIS
LIN {X 0.132,Y -562.769,Z 945.278,A 0.000,B 0.000,C 90.000,E1 86.045} C_DIS
LIN {X 0.273,Y -562.991,Z 945.269,A 0.000,B 0.000,C 90.000,E1 84.375} C_DIS
LIN {X 0.037,Y -563.138,Z 945.264,A 0.000,B 0.000,C 90.000,E1 83.571} C_DIS
LIN {X 0.257,Y -563.413,Z 945.255,A 0.000,B 0.000,C 90.000,E1 81.894} C_DIS
LIN {X -0.144,Y -564.254,Z 945.241,A 0.000,B 0.000,C 90.000,E1 79.454} C_DIS
LIN {X 0.132,Y -564.890,Z 945.234,A 0.000,B 0.000,C 90.000,E1 78.049} C_DIS
LIN {X -0.179,Y -566.199,Z 945.221,A 0.000,B 0.000,C 90.000,E1 75.880} C_DIS
LIN {X 0.190,Y -567.343,Z 945.211,A 0.000,B 0.000,C 90.000,E1 73.921} C_DIS
LIN {X 0.251,Y -568.247,Z 945.203,A 0.000,B 0.000,C 90.000,E1 72.543} C_DIS
LIN {X -0.259,Y -569.263,Z 945.193,A 0.000,B 0.000,C 90.000,E1 70.678} C_DIS
LIN {X 0.044,Y -569.651,Z 945.188,A 0.000,B 0.000,C 90.000,E1 69.826} C_DIS
LIN {X 0.336,Y -570.200,Z 945.179,A 0.000,B 0.000,C 90.000,E1 68.156} C_DIS
LIN {X -0.279,Y -570.669,Z 945.168,A 0.000,B 0.000,C 90.000,E1 66.305} C_DIS
LIN {X -0.263,Y -571.016,Z 945.159,A 0.000,B 0.000,C 90.000,E1 64.665} C_DIS
LIN {X 0.176,Y -571.188,Z 945.152,A 0.000,B 0.000,C 90.000,E1 63.256} C_DIS
LIN {X 0.113,Y -571.336,Z 945.144,A 0.000,B 0.000,C 90.000,E1 61.897} C_DIS
LIN {X -0.011,Y -571.402,Z 945.133,A 0.000,B 0.000,C 90.000,E1 59.999} C_DIS
LIN {X 0.198,Y -571.520,Z 945.126,A 0.000,B 0.000,C 90.000,E1 58.614} C_DIS
LIN {X 0.037,Y -571.301,Z 945.117,A 0.000,B 0.000,C 90.000,E1 56.993} C_DIS
LIN {X -0.292,Y -570.746,Z 945.108,A 0.000,B 0.000,C 90.000,E1 55.388} C_DIS
LIN {X 0.036,Y -570.209,Z 945.100,A 0.000,B 0.000,C 90.000,E1 53.989} C_DIS
LIN {X -0.240,Y -569.432,Z 945.094,A 0.000,B 0.000,C 90.000,E1 52.924} C_DIS
LIN {X -0.181,Y -568.472,Z 945.088,A 0.000,B 0.000,C 90.000,E1 51.823} C_DIS
LIN {X 0.189,Y -567.639,Z 945.083,A 0.000,B 0.000,C 90.000,E1 50.964} C_DIS
LIN {X 0.103,Y -566.698,Z 945.079,A 0.000,B 0.000,C 90.000,E1 50.150} C_DIS
LIN {X 0.056,Y -565.118,Z 945.073,A 0.000,B 0.000,C 90.000,E1 49.057} C_DIS
LIN {X -0.157,Y -564.281,Z 945.070,A 0.000,B 0.000,C 90.000,E1 48.528} C_DIS
LIN {X 0.189,Y -562.177,Z 945.063,A 0.000,B 0.000,C 90.000,E1 47.391} C_DIS
LIN {X -0.051,Y -561.054,Z 945.060,A 0.000,B 0.000,C 90.000,E1 46.863} C_DIS
LIN {X 0.215,Y -558.377,Z 945.054,A 0.000,B 0.000,C 90.000,E1 45.729} C_DIS
LIN {X -0.058,Y -556.893,Z 945.051,A 0.000,B 0.000,C 90.000,E1 45.202} C_DIS
LIN {X 0.102,Y -554.397,Z 945.047,A 0.000,B 0.000,C 90.000,E1 44.352} C_DIS
LIN {X 0.193,Y -552.565,Z 945.043,A 0.000,B 0.000,C 90.000,E1 43.785} C_DIS
LIN {X -0.090,Y -549.544,Z 945.039,A 0.000,B 0.000,C 90.000,E1 42.975} C_DIS
LIN {X -0.005,Y -547.346,Z 945.036,A 0.000,B 0.000,C 90.000,E1 42.405} C_DIS
LIN {X -0.149,Y -543.138,Z 945.030,A 0.000,B 0.000,C 90.000,E1 41.434} C_DIS
LIN {X 0.102,Y -538.162,Z 945.025,A 0.000,B 0.000,C 90.000,E1 40.415} C_DIS
LIN {X -0.120,Y -535.916,Z 945.022,A 0.000,B 0.000,C 90.000,E1 40.011} C_DIS
LIN {X 0.051,Y -531.812,Z 945.018,A 0.000,B 0.000,C 90.000,E1 39.277} C_DIS
LIN {X 0.161,Y -525.825,Z 945.013,A 0.000,B 0.000,C 90.000,E1 38.257} C_DIS
LIN {X 0.237,Y -521.287,Z 945.009,A 0.000,B 0.000,C 90.000,E1 37.523} C_DIS
LIN {X 0.010,Y -518.469,Z 945.006,A 0.000,B 0.000,C 90.000,E1 37.111} C_DIS
LIN {X -0.053,Y -511.441,Z 945.001,A 0.000,B 0.000,C 90.000,E1 36.091} C_DIS
LIN {X 0.295,Y -506.069,Z 944.996,A 0.000,B 0.000,C 90.000,E1 35.311} C_DIS
LIN {X -0.002,Y -502.665,Z 944.994,A 0.000,B 0.000,C 90.000,E1 34.898} C_DIS
LIN {X 0.031,Y -498.064,Z 944.991,A 0.000,B 0.000,C 90.000,E1 34.326} C_DIS
LIN {X 0.193,Y -492.823,Z 944.987,A 0.000,B 0.000,C 90.000,E1 33.706} C_DIS
LIN {X -0.066,Y -486.106,Z 944.983,A 0.000,B 0.000,C 90.000,E1 33.007} C_DIS
LIN {X 0.277,Y -477.799,Z 944.979,A 0.000,B 0.000,C 90.000,E1 32.133} C_DIS
LIN {X 0.031,Y -469.027,Z 944.974,A 0.000,B 0.000,C 90.000,E1 31.337} C_DIS
LIN {X -0.028,Y -461.627,Z 944.970,A 0.000,B 0.000,C 90.000,E1 30.669} C_DIS
LIN {X 0.073,Y -451.101,Z 944.965,A 0.000,B 0.000,C 90.000,E1 29.745} C_DIS
LIN {X 0.167,Y -443.321,Z 944.962,A 0.000,B 0.000,C 90.000,E1 29.077} C_DIS
LIN {X 0.276,Y -428.147,Z 944.955,A 0.000,B 0.000,C 90.000,E1 27.769} C_DIS
LIN {X 0.144,Y -408.669,Z 944.944,A 0.000,B 0.000,C 90.000,E1 25.976} C_DIS
LIN {X 0.079,Y -398.635,Z 944.939,A 0.000,B 0.000,C 90.000,E1 24.951} C_DIS
LIN {X -0.004,Y -394.901,Z 944.936,A 0.000,B 0.000,C 90.000,E1 24.515} C_DIS
LIN {X 0.045,Y -392.878,Z 944.935,A 0.000,B 0.000,C 90.000,E1 24.207} C_DIS
LIN {X 0.044,Y -390.471,Z 944.931,A 0.000,B 0.000,C 90.000,E1 23.643} C_DIS
LIN {X -0.118,Y -389.470,Z 944.928,A 0.000,B 0.000,C 90.000,E1 23.131} C_DIS
LIN {X 0.246,Y -389.157,Z 944.925,A 0.000,B 0.000,C 90.000,E1 22.514} C_DIS
LIN {X -0.003,Y -389.354,Z 944.921,A 0.000,B 0.000,C 90.000,E1 21.844} C_DIS
LIN {X -0.075,Y -393.218,Z 944.898,A 0.000,B 0.000,C 90.000,E1 17.583} C_DIS
LIN {X 0.168,Y -396.564,Z 944.882,A 0.000,B 0.000,C 90.000,E1 14.717} C_DIS
LIN {X -0.120,Y -399.459,Z 944.870,A 0.000,B 0.000,C 90.000,E1 12.647} C_DIS
LIN {X -0.132,Y -404.347,Z 944.853,A 0.000,B 0.000,C 90.000,E1 9.500} C_DIS
LIN {X -0.087,Y -407.947,Z 944.841,A 0.000,B 0.000,C 90.000,E1 7.409} C_DIS
LIN {X -0.081,Y -412.498,Z 944.828,A 0.000,B 0.000,C 90.000,E1 4.992} C_DIS
LIN {X 0.047,Y -418.248,Z 944.813,A 0.000,B 0.000,C 90.000,E1 2.236} C_DIS
LIN {X -0.167,Y -425.801,Z 944.795,A 0.000,B 0.000,C 90.000,E1 359.141} C_DIS
LIN {X 0.007,Y -428.193,Z 944.791,A 0.000,B 0.000,C 90.000,E1 358.453} C_DIS
LIN {X 0.081,Y -429.870,Z 944.790,A 0.000,B 0.000,C 90.000,E1 358.108} C_DIS
LIN {X 0.117,Y -430.798,Z 944.789,A 0.000,B 0.000,C 90.000,E1 357.936} C_DIS
LIN {X 0.152,Y -431.957,Z 944.788,A 0.000,B 0.000,C 90.000,E1 357.764} C_DIS
LIN {X -0.099,Y -434.786,Z 944.786,A 0.000,B 0.000,C 90.000,E1 357.478} C_DIS
LIN {X 0.010,Y -436.399,Z 944.785,A 0.000,B 0.000,C 90.000,E1 357.306} C_DIS
LIN {X 0.208,Y -440.109,Z 944.784,A 0.000,B 0.000,C 90.000,E1 357.020} C_DIS
LIN {X -0.019,Y -449.618,Z 944.781,A 0.000,B 0.000,C 90.000,E1 356.560} C_DIS
LIN {X -0.144,Y -461.429,Z 944.778,A 0.000,B 0.000,C 90.000,E1 355.988} C_DIS
LIN {X -0.205,Y -471.389,Z 944.775,A 0.000,B 0.000,C 90.000,E1 355.469} C_DIS
LIN {X -0.223,Y -481.378,Z 944.772,A 0.000,B 0.000,C 90.000,E1 354.951} C_DIS
LIN {X 0.201,Y -494.352,Z 944.768,A 0.000,B 0.000,C 90.000,E1 354.204} C_DIS
LIN {X -0.218,Y -507.176,Z 944.764,A 0.000,B 0.000,C 90.000,E1 353.514} C_DIS
LIN {X -0.179,Y -518.351,Z 944.760,A 0.000,B 0.000,C 90.000,E1 352.818} C_DIS
LIN {X -0.197,Y -526.021,Z 944.757,A 0.000,B 0.000,C 90.000,E1 352.299} C_DIS
LIN {X 0.018,Y -533.545,Z 944.754,A 0.000,B 0.000,C 90.000,E1 351.724} C_DIS
LIN {X 0.005,Y -540.731,Z 944.751,A 0.000,B 0.000,C 90.000,E1 351.141} C_DIS
LIN {X -0.288,Y -546.371,Z 944.748,A 0.000,B 0.000,C 90.000,E1 350.679} C_DIS
LIN {X -0.128,Y -551.585,Z 944.745,A 0.000,B 0.000,C 90.000,E1 350.151} C_DIS
LIN {X 0.138,Y -557.932,Z 944.742,A 0.000,B 0.000,C 90.000,E1 349.454} C_DIS
LIN {X 0.204,Y -563.821,Z 944.738,A 0.000,B 0.000,C 90.000,E1 348.757} C_DIS
LIN {X 0.228,Y -567.202,Z 944.735,A 0.000,B 0.000,C 90.000,E1 348.342} C_DIS
LIN {X -0.029,Y -574.256,Z 944.730,A 0.000,B 0.000,C 90.000,E1 347.409} C_DIS
LIN {X 0.267,Y -578.967,Z 944.726,A 0.000,B 0.000,C 90.000,E1 346.700} C_DIS
LIN {X -0.051,Y -586.531,Z 944.720,A 0.000,B 0.000,C 90.000,E1 345.519} C_DIS
LIN {X -0.263,Y -593.256,Z 944.713,A 0.000,B 0.000,C 90.000,E1 344.338} C_DIS
LIN {X 0.202,Y -596.749,Z 944.709,A 0.000,B 0.000,C 90.000,E1 343.630} C_DIS
LIN {X -0.043,Y -601.955,Z 944.703,A 0.000,B 0.000,C 90.000,E1 342.598} C_DIS
LIN {X 0.138,Y -607.509,Z 944.697,A 0.000,B 0.000,C 90.000,E1 341.402} C_DIS
LIN {X 0.070,Y -611.630,Z 944.692,A 0.000,B 0.000,C 90.000,E1 340.496} C_DIS
LIN {X 0.280,Y -614.937,Z 944.687,A 0.000,B 0.000,C 90.000,E1 339.699} C_DIS
LIN {X -0.300,Y -619.155,Z 944.682,A 0.000,B 0.000,C 90.000,E1 338.720} C_DIS
LIN {X -0.023,Y -623.095,Z 944.676,A 0.000,B 0.000,C 90.000,E1 337.667} C_DIS
LIN {X -0.263,Y -626.805,Z 944.670,A 0.000,B 0.000,C 90.000,E1 336.666} C_DIS
LIN {X 0.119,Y -630.245,Z 944.665,A 0.000,B 0.000,C 90.000,E1 335.613} C_DIS
LIN {X -0.001,Y -634.213,Z 944.658,A 0.000,B 0.000,C 90.000,E1 334.357} C_DIS
LIN {X -0.351,Y -637.954,Z 944.651,A 0.000,B 0.000,C 90.000,E1 333.127} C_DIS
LIN {X -0.129,Y -640.645,Z 944.645,A 0.000,B 0.000,C 90.000,E1 332.103} C_DIS
LIN {X 0.365,Y -642.554,Z 944.641,A 0.000,B 0.000,C 90.000,E1 331.307} C_DIS
LIN {X -0.335,Y -645.999,Z 944.633,A 0.000,B 0.000,C 90.000,E1 329.871} C_DIS
LIN {X -0.181,Y -648.564,Z 944.626,A 0.000,B 0.000,C 90.000,E1 328.614} C_DIS
LIN {X 0.272,Y -650.335,Z 944.620,A 0.000,B 0.000,C 90.000,E1 327.582} C_DIS
LIN {X -0.144,Y -651.900,Z 944.615,A 0.000,B 0.000,C 90.000,E1 326.628} C_DIS
LIN {X -0.096,Y -653.593,Z 944.608,A 0.000,B 0.000,C 90.000,E1 325.388} C_DIS
LIN {X -0.028,Y -654.530,Z 944.604,A 0.000,B 0.000,C 90.000,E1 324.642} C_DIS
LIN {X -0.101,Y -655.760,Z 944.597,A 0.000,B 0.000,C 90.000,E1 323.417} C_DIS
LIN {X -0.144,Y -656.825,Z 944.590,A 0.000,B 0.000,C 90.000,E1 322.190} C_DIS
LIN {X -0.220,Y -657.948,Z 944.582,A 0.000,B 0.000,C 90.000,E1 320.723} C_DIS
LIN {X -0.287,Y -658.721,Z 944.576,A 0.000,B 0.000,C 90.000,E1 319.747} C_DIS
LIN {X 0.043,Y -660.031,Z 944.565,A 0.000,B 0.000,C 90.000,E1 317.757} C_DIS
LIN {X -0.049,Y -661.228,Z 944.557,A 0.000,B 0.000,C 90.000,E1 316.296} C_DIS
LIN {X -0.115,Y -662.016,Z 944.552,A 0.000,B 0.000,C 90.000,E1 315.324} C_DIS
LIN {X 0.247,Y -664.166,Z 944.538,A 0.000,B 0.000,C 90.000,E1 312.852} C_DIS
LIN {X 0.242,Y -665.552,Z 944.530,A 0.000,B 0.000,C 90.000,E1 311.391} C_DIS
LIN {X 0.267,Y -666.640,Z 944.523,A 0.000,B 0.000,C 90.000,E1 310.172} C_DIS
LIN {X -0.133,Y -667.855,Z 944.515,A 0.000,B 0.000,C 90.000,E1 308.749} C_DIS
LIN {X 0.019,Y -668.714,Z 944.509,A 0.000,B 0.000,C 90.000,E1 307.523} C_DIS
LIN {X -0.330,Y -669.219,Z 944.503,A 0.000,B 0.000,C 90.000,E1 306.583} C_DIS
LIN {X -0.035,Y -669.699,Z 944.495,A 0.000,B 0.000,C 90.000,E1 305.105} C_DIS
LIN {X -0.422,Y -670.522,Z 944.483,A 0.000,B 0.000,C 90.000,E1 302.959} C_DIS
LIN {X 0.080,Y -671.253,Z 944.475,A 0.000,B 0.000,C 90.000,E1 301.465} C_DIS
LIN {X -0.193,Y -675.186,Z 944.452,A 0.000,B 0.000,C 90.000,E1 297.385} C_DIS
LIN {X -0.210,Y -678.358,Z 944.441,A 0.000,B 0.000,C 90.000,E1 295.463} C_DIS
LIN {X -0.140,Y -680.327,Z 944.435,A 0.000,B 0.000,C 90.000,E1 294.259} C_DIS
LIN {X 0.379,Y -681.727,Z 944.429,A 0.000,B 0.000,C 90.000,E1 293.259} C_DIS
LIN {X -0.179,Y -682.390,Z 944.425,A 0.000,B 0.000,C 90.000,E1 292.589} C_DIS
LIN {X 0.022,Y -682.301,Z 944.424,A 0.000,B 0.000,C 90.000,E1 292.333} C_DIS
LIN {X 0.164,Y -681.687,Z 944.422,A 0.000,B 0.000,C 90.000,E1 291.844} C_DIS
LIN {X 0.361,Y -680.682,Z 944.420,A 0.000,B 0.000,C 90.000,E1 291.589} C_DIS
LIN {X -0.231,Y -678.826,Z 944.418,A 0.000,B 0.000,C 90.000,E1 291.280} C_DIS
LIN {X -0.138,Y -678.073,Z 944.417,A 0.000,B 0.000,C 90.000,E1 291.153} C_DIS
LIN {X -0.290,Y -676.964,Z 944.417,A 0.000,B 0.000,C 90.000,E1 291.046} C_DIS
LIN {X 0.275,Y -672.712,Z 944.415,A 0.000,B 0.000,C 90.000,E1 290.663} C_DIS
LIN {X 0.088,Y -667.919,Z 944.413,A 0.000,B 0.000,C 90.000,E1 290.375} C_DIS
LIN {X 0.021,Y -663.890,Z 944.412,A 0.000,B 0.000,C 90.000,E1 290.120} C_DIS
LIN {X 0.043,Y -661.439,Z 944.411,A 0.000,B 0.000,C 90.000,E1 289.939} C_DIS
LIN {X 0.007,Y -661.406,Z 944.411,A 0.000,B 0.000,C 90.000,E1 289.939} C_DIS
LIN {X 0.257,Y -660.846,Z 944.410,A 0.000,B 0.000,C 90.000,E1 289.812} C_DIS
LIN {X 0.106,Y -661.095,Z 944.408,A 0.000,B 0.000,C 90.000,E1 289.504} C_DIS
LIN {X -0.054,Y -662.719,Z 944.406,A 0.000,B 0.000,C 90.000,E1 289.033} C_DIS
LIN {X -0.176,Y -670.472,Z 944.398,A 0.000,B 0.000,C 90.000,E1 287.583} C_DIS
LIN {X -0.120,Y -672.855,Z 944.395,A 0.000,B 0.000,C 90.000,E1 287.094} C_DIS
LIN {X -0.117,Y -675.926,Z 944.391,A 0.000,B 0.000,C 90.000,E1 286.370} C_DIS
LIN {X -0.226,Y -677.641,Z 944.388,A 0.000,B 0.000,C 90.000,E1 285.898} C_DIS
LIN {X -0.363,Y -679.767,Z 944.384,A 0.000,B 0.000,C 90.000,E1 285.190} C_DIS
LIN {X 0.184,Y -681.410,Z 944.380,A 0.000,B 0.000,C 90.000,E1 284.426} C_DIS
LIN {X 0.063,Y -683.239,Z 944.375,A 0.000,B 0.000,C 90.000,E1 283.480} C_DIS
LIN {X -0.014,Y -684.291,Z 944.371,A 0.000,B 0.000,C 90.000,E1 282.771} C_DIS
LIN {X -0.109,Y -685.340,Z 944.366,A 0.000,B 0.000,C 90.000,E1 281.827} C_DIS
LIN {X -0.292,Y -685.549,Z 944.363,A 0.000,B 0.000,C 90.000,E1 281.366} C_DIS
LIN {X 0.312,Y -685.446,Z 944.359,A 0.000,B 0.000,C 90.000,E1 280.602} C_DIS
LIN {X 0.140,Y -685.028,Z 944.356,A 0.000,B 0.000,C 90.000,E1 280.141} C_DIS
LIN {X 0.084,Y -684.150,Z 944.354,A 0.000,B 0.000,C 90.000,E1 279.670} C_DIS
LIN {X -0.092,Y -682.974,Z 944.351,A 0.000,B 0.000,C 90.000,E1 279.208} C_DIS
LIN {X -0.127,Y -682.289,Z 944.350,A 0.000,B 0.000,C 90.000,E1 278.973} C_DIS
LIN {X -0.312,Y -680.599,Z 944.347,A 0.000,B 0.000,C 90.000,E1 278.511} C_DIS
LIN {X 0.169,Y -678.513,Z 944.345,A 0.000,B 0.000,C 90.000,E1 277.992} C_DIS
LIN {X -0.248,Y -673.803,Z 944.339,A 0.000,B 0.000,C 90.000,E1 277.068} C_DIS
LIN {X 0.102,Y -669.815,Z 944.335,A 0.000,B 0.000,C 90.000,E1 276.315} C_DIS
LIN {X -0.245,Y -666.006,Z 944.332,A 0.000,B 0.000,C 90.000,E1 275.739} C_DIS
LIN {X 0.131,Y -662.536,Z 944.329,A 0.000,B 0.000,C 90.000,E1 275.220} C_DIS
LIN {X -0.179,Y -658.706,Z 944.326,A 0.000,B 0.000,C 90.000,E1 274.759} C_DIS
LIN {X -0.008,Y -653.250,Z 944.323,A 0.000,B 0.000,C 90.000,E1 274.131} C_DIS
LIN {X 0.274,Y -648.579,Z 944.320,A 0.000,B 0.000,C 90.000,E1 273.612} C_DIS
LIN {X -0.092,Y -643.658,Z 944.318,A 0.000,B 0.000,C 90.000,E1 273.154} C_DIS
LIN {X -0.259,Y -637.011,Z 944.314,A 0.000,B 0.000,C 90.000,E1 272.579} C_DIS
LIN {X -0.194,Y -631.531,Z 944.312,A 0.000,B 0.000,C 90.000,E1 272.121} C_DIS
LIN {X 0.143,Y -625.614,Z 944.309,A 0.000,B 0.000,C 90.000,E1 271.661} C_DIS
LIN {X -0.298,Y -618.108,Z 944.307,A 0.000,B 0.000,C 90.000,E1 271.203} C_DIS
LIN {X 0.166,Y -610.347,Z 944.304,A 0.000,B 0.000,C 90.000,E1 270.688} C_DIS
LIN {X 0.056,Y -603.767,Z 944.302,A 0.000,B 0.000,C 90.000,E1 270.344} C_DIS
LIN {X 0.195,Y -597.029,Z 944.300,A 0.000,B 0.000,C 90.000,E1 270.000} C_DIS
LIN {X 0.080,Y -589.874,Z 944.299,A 0.000,B 0.000,C 90.000,E1 269.714} C_DIS
LIN {X -0.216,Y -584.544,Z 944.297,A 0.000,B 0.000,C 90.000,E1 269.542} C_DIS
LIN {X 0.255,Y -578.463,Z 944.296,A 0.000,B 0.000,C 90.000,E1 269.312} C_DIS
LIN {X 0.074,Y -570.766,Z 944.295,A 0.000,B 0.000,C 90.000,E1 269.141} C_DIS
LIN {X 0.049,Y -564.513,Z 944.295,A 0.000,B 0.000,C 90.000,E1 269.026} C_DIS
LIN {X -0.020,Y -559.231,Z 944.294,A 0.000,B 0.000,C 90.000,E1 268.969} C_DIS
LIN {X 0.195,Y -553.901,Z 944.294,A 0.000,B 0.000,C 90.000,E1 268.912} C_DIS
LIN {X -0.122,Y -549.894,Z 944.294,A 0.000,B 0.000,C 90.000,E1 268.912} C_DIS
LIN {X 0.195,Y -548.409,Z 944.294,A 0.000,B 0.000,C 90.000,E1 268.854} C_DIS
LIN {X -0.258,Y -547.255,Z 944.294,A 0.000,B 0.000,C 90.000,E1 268.854} C_DIS
LIN {X 0.018,Y -544.421,Z 944.293,A 0.000,B 0.000,C 90.000,E1 268.682} C_DIS
LIN {X -0.036,Y -544.284,Z 944.293,A 0.000,B 0.000,C 90.000,E1 268.682} C_DIS
LIN {X -0.073,Y -543.817,Z 944.292,A 0.000,B 0.000,C 90.000,E1 268.511} C_DIS
LIN {X 0.117,Y -540.635,Z 944.273,A 0.000,B 0.000,C 90.000,E1 265.065} C_DIS
LIN {X -0.273,Y -539.652,Z 944.265,A 0.000,B 0.000,C 90.000,E1 263.685} C_DIS
LIN {X -0.026,Y -538.485,Z 944.255,A 0.000,B 0.000,C 90.000,E1 261.951} C_DIS
LIN {X 0.087,Y -537.839,Z 944.251,A 0.000,B 0.000,C 90.000,E1 261.084} C_DIS
LIN {X 0.187,Y -536.954,Z 944.246,A 0.000,B 0.000,C 90.000,E1 260.218} C_DIS
LIN {X -0.102,Y -535.434,Z 944.239,A 0.000,B 0.000,C 90.000,E1 259.106} C_DIS
LIN {X -0.255,Y -532.747,Z 944.228,A 0.000,B 0.000,C 90.000,E1 257.117} C_DIS
LIN {X 0.284,Y -530.393,Z 944.217,A 0.000,B 0.000,C 90.000,E1 255.046} C_DIS
LIN {X 0.225,Y -528.389,Z 944.208,A 0.000,B 0.000,C 90.000,E1 253.323} C_DIS
LIN {X 0.099,Y -526.682,Z 944.200,A 0.000,B 0.000,C 90.000,E1 251.891} C_DIS
LIN {X 0.273,Y -524.830,Z 944.191,A 0.000,B 0.000,C 90.000,E1 250.423} C_DIS
LIN {X -0.093,Y -522.584,Z 944.182,A 0.000,B 0.000,C 90.000,E1 248.720} C_DIS
LIN {X 0.051,Y -521.103,Z 944.175,A 0.000,B 0.000,C 90.000,E1 247.539} C_DIS
LIN {X -0.012,Y -518.502,Z 944.166,A 0.000,B 0.000,C 90.000,E1 245.793} C_DIS
LIN {X 0.078,Y -515.712,Z 944.156,A 0.000,B 0.000,C 90.000,E1 244.024} C_DIS
LIN {X -0.129,Y -512.908,Z 944.146,A 0.000,B 0.000,C 90.000,E1 242.281} C_DIS
LIN {X -0.043,Y -510.519,Z 944.138,A 0.000,B 0.000,C 90.000,E1 240.795} C_DIS
LIN {X -0.170,Y -508.956,Z 944.133,A 0.000,B 0.000,C 90.000,E1 239.921} C_DIS
LIN {X 0.081,Y -506.228,Z 944.125,A 0.000,B 0.000,C 90.000,E1 238.408} C_DIS
LIN {X 0.104,Y -503.010,Z 944.116,A 0.000,B 0.000,C 90.000,E1 236.914} C_DIS
LIN {X -0.068,Y -499.598,Z 944.108,A 0.000,B 0.000,C 90.000,E1 235.435} C_DIS
LIN {X 0.099,Y -494.167,Z 944.095,A 0.000,B 0.000,C 90.000,E1 233.004} C_DIS
LIN {X 0.206,Y -490.151,Z 944.084,A 0.000,B 0.000,C 90.000,E1 231.170} C_DIS
LIN {X -0.126,Y -487.399,Z 944.078,A 0.000,B 0.000,C 90.000,E1 229.989} C_DIS
LIN {X -0.044,Y -483.886,Z 944.069,A 0.000,B 0.000,C 90.000,E1 228.447} C_DIS
LIN {X 0.019,Y -478.329,Z 944.055,A 0.000,B 0.000,C 90.000,E1 225.972} C_DIS
LIN {X 0.020,Y -474.147,Z 944.045,A 0.000,B 0.000,C 90.000,E1 224.109} C_DIS
LIN {X 0.084,Y -471.403,Z 944.038,A 0.000,B 0.000,C 90.000,E1 222.852} C_DIS
LIN {X -0.130,Y -468.012,Z 944.029,A 0.000,B 0.000,C 90.000,E1 221.310} C_DIS
LIN {X 0.150,Y -462.482,Z 944.015,A 0.000,B 0.000,C 90.000,E1 218.749} C_DIS
LIN {X -0.081,Y -458.312,Z 944.005,A 0.000,B 0.000,C 90.000,E1 216.870} C_DIS
LIN {X 0.231,Y -454.766,Z 943.996,A 0.000,B 0.000,C 90.000,E1 215.231} C_DIS
LIN {X 0.291,Y -450.553,Z 943.985,A 0.000,B 0.000,C 90.000,E1 213.293} C_DIS
LIN {X 0.237,Y -447.640,Z 943.978,A 0.000,B 0.000,C 90.000,E1 212.005} C_DIS
LIN {X -0.023,Y -444.110,Z 943.969,A 0.000,B 0.000,C 90.000,E1 210.413} C_DIS
LIN {X 0.085,Y -439.882,Z 943.958,A 0.000,B 0.000,C 90.000,E1 208.437} C_DIS
LIN {X 0.053,Y -436.329,Z 943.949,A 0.000,B 0.000,C 90.000,E1 206.796} C_DIS
LIN {X -0.056,Y -432.662,Z 943.940,A 0.000,B 0.000,C 90.000,E1 205.155} C_DIS
LIN {X 0.165,Y -429.006,Z 943.931,A 0.000,B 0.000,C 90.000,E1 203.462} C_DIS
LIN {X -0.051,Y -425.998,Z 943.923,A 0.000,B 0.000,C 90.000,E1 202.153} C_DIS
LIN {X -0.171,Y -420.859,Z 943.910,A 0.000,B 0.000,C 90.000,E1 199.812} C_DIS
LIN {X -0.168,Y -415.300,Z 943.895,A 0.000,B 0.000,C 90.000,E1 197.094} C_DIS
LIN {X -0.074,Y -411.863,Z 943.885,A 0.000,B 0.000,C 90.000,E1 195.371} C_DIS
LIN {X -0.167,Y -409.079,Z 943.878,A 0.000,B 0.000,C 90.000,E1 194.008} C_DIS
LIN {X 0.200,Y -404.246,Z 943.864,A 0.000,B 0.000,C 90.000,E1 191.535} C_DIS
LIN {X -0.193,Y -400.926,Z 943.855,A 0.000,B 0.000,C 90.000,E1 189.849} C_DIS
LIN {X 0.144,Y -397.588,Z 943.845,A 0.000,B 0.000,C 90.000,E1 188.049} C_DIS
LIN {X -0.044,Y -394.202,Z 943.835,A 0.000,B 0.000,C 90.000,E1 186.315} C_DIS
LIN {X -0.038,Y -390.291,Z 943.823,A 0.000,B 0.000,C 90.000,E1 184.188} C_DIS
LIN {X 0.054,Y -385.585,Z 943.807,A 0.000,B 0.000,C 90.000,E1 181.318} C_DIS
LIN {X 0.130,Y -384.281,Z 943.801,A 0.000,B 0.000,C 90.000,E1 180.229} C_DIS
LIN {X -0.083,Y -383.709,Z 943.797,A 0.000,B 0.000,C 90.000,E1 179.542} C_DIS
LIN {X 0.081,Y -383.465,Z 943.793,A 0.000,B 0.000,C 90.000,E1 178.797} C_DIS
LIN {X -0.130,Y -383.861,Z 943.789,A 0.000,B 0.000,C 90.000,E1 178.108} C_DIS
LIN {X 0.052,Y -385.319,Z 943.784,A 0.000,B 0.000,C 90.000,E1 177.192} C_DIS
LIN {X -0.003,Y -385.753,Z 943.784,A 0.000,B 0.000,C 90.000,E1 177.020} C_DIS
LIN {X -0.067,Y -388.093,Z 943.780,A 0.000,B 0.000,C 90.000,E1 176.445} C_DIS
LIN {X -0.117,Y -388.987,Z 943.779,A 0.000,B 0.000,C 90.000,E1 176.274} C_DIS
LIN {X -0.040,Y -391.982,Z 943.777,A 0.000,B 0.000,C 90.000,E1 175.812} C_DIS
LIN {X -0.016,Y -394.790,Z 943.775,A 0.000,B 0.000,C 90.000,E1 175.469} C_DIS
LIN {X 0.022,Y -398.609,Z 943.773,A 0.000,B 0.000,C 90.000,E1 175.065} C_DIS
LIN {X 0.116,Y -414.070,Z 943.765,A 0.000,B 0.000,C 90.000,E1 173.742} C_DIS
LIN {X 0.209,Y -424.583,Z 943.761,A 0.000,B 0.000,C 90.000,E1 172.875} C_DIS
LIN {X -0.197,Y -435.369,Z 943.755,A 0.000,B 0.000,C 90.000,E1 172.008} C_DIS
LIN {X 0.155,Y -441.488,Z 943.753,A 0.000,B 0.000,C 90.000,E1 171.432} C_DIS
LIN {X 0.061,Y -450.345,Z 943.748,A 0.000,B 0.000,C 90.000,E1 170.622} C_DIS
LIN {X -0.030,Y -459.060,Z 943.743,A 0.000,B 0.000,C 90.000,E1 169.803} C_DIS
LIN {X 0.105,Y -467.487,Z 943.739,A 0.000,B 0.000,C 90.000,E1 168.926} C_DIS
LIN {X 0.181,Y -477.035,Z 943.733,A 0.000,B 0.000,C 90.000,E1 167.881} C_DIS
LIN {X -0.101,Y -480.788,Z 943.730,A 0.000,B 0.000,C 90.000,E1 167.465} C_DIS
LIN {X 0.085,Y -485.788,Z 943.727,A 0.000,B 0.000,C 90.000,E1 166.825} C_DIS
LIN {X 0.099,Y -488.369,Z 943.725,A 0.000,B 0.000,C 90.000,E1 166.520} C_DIS
LIN {X -0.167,Y -495.398,Z 943.720,A 0.000,B 0.000,C 90.000,E1 165.644} C_DIS
LIN {X -0.189,Y -499.844,Z 943.717,A 0.000,B 0.000,C 90.000,E1 165.046} C_DIS
LIN {X 0.010,Y -507.275,Z 943.711,A 0.000,B 0.000,C 90.000,E1 163.976} C_DIS
LIN {X -0.157,Y -512.135,Z 943.707,A 0.000,B 0.000,C 90.000,E1 163.251} C_DIS
LIN {X 0.061,Y -517.242,Z 943.703,A 0.000,B 0.000,C 90.000,E1 162.489} C_DIS
LIN {X 0.025,Y -521.801,Z 943.699,A 0.000,B 0.000,C 90.000,E1 161.764} C_DIS
LIN {X 0.040,Y -524.735,Z 943.696,A 0.000,B 0.000,C 90.000,E1 161.329} C_DIS
LIN {X 0.036,Y -531.070,Z 943.691,A 0.000,B 0.000,C 90.000,E1 160.315} C_DIS
LIN {X 0.139,Y -538.192,Z 943.684,A 0.000,B 0.000,C 90.000,E1 159.156} C_DIS
LIN {X -0.079,Y -543.330,Z 943.680,A 0.000,B 0.000,C 90.000,E1 158.337} C_DIS
LIN {X 0.204,Y -550.150,Z 943.673,A 0.000,B 0.000,C 90.000,E1 157.177} C_DIS
LIN {X 0.117,Y -554.152,Z 943.669,A 0.000,B 0.000,C 90.000,E1 156.485} C_DIS
LIN {X -0.144,Y -559.603,Z 943.664,A 0.000,B 0.000,C 90.000,E1 155.537} C_DIS
LIN {X 0.073,Y -565.337,Z 943.658,A 0.000,B 0.000,C 90.000,E1 154.409} C_DIS
LIN {X -0.300,Y -568.115,Z 943.655,A 0.000,B 0.000,C 90.000,E1 153.896} C_DIS
LIN {X 0.286,Y -573.419,Z 943.649,A 0.000,B 0.000,C 90.000,E1 152.743} C_DIS
LIN {X -0.143,Y -578.858,Z 943.642,A 0.000,B 0.000,C 90.000,E1 151.563} C_DIS
LIN {X 0.078,Y -583.457,Z 943.636,A 0.000,B 0.000,C 90.000,E1 150.461} C_DIS
LIN {X 0.025,Y -588.766,Z 943.629,A 0.000,B 0.000,C 90.000,E1 149.125} C_DIS
LIN {X -0.137,Y -592.789,Z 943.623,A 0.000,B 0.000,C 90.000,E1 148.074} C_DIS
LIN {X 0.282,Y -597.613,Z 943.615,A 0.000,B 0.000,C 90.000,E1 146.707} C_DIS
LIN {X 0.292,Y -602.337,Z 943.608,A 0.000,B 0.000,C 90.000,E1 145.388} C_DIS
LIN {X 0.158,Y -607.820,Z 943.599,A 0.000,B 0.000,C 90.000,E1 143.829} C_DIS
LIN {X 0.131,Y -613.193,Z 943.591,A 0.000,B 0.000,C 90.000,E1 142.271} C_DIS
LIN {X 0.102,Y -618.649,Z 943.582,A 0.000,B 0.000,C 90.000,E1 140.723} C_DIS
LIN {X -0.145,Y -623.077,Z 943.575,A 0.000,B 0.000,C 90.000,E1 139.461} C_DIS
LIN {X -0.064,Y -632.553,Z 943.561,A 0.000,B 0.000,C 90.000,E1 136.905} C_DIS
LIN {X -0.232,Y -638.247,Z 943.552,A 0.000,B 0.000,C 90.000,E1 135.405} C_DIS
LIN {X 0.237,Y -642.953,Z 943.545,A 0.000,B 0.000,C 90.000,E1 134.109} C_DIS
LIN {X 0.212,Y -649.490,Z 943.536,A 0.000,B 0.000,C 90.000,E1 132.366} C_DIS
LIN {X -0.065,Y -655.113,Z 943.527,A 0.000,B 0.000,C 90.000,E1 130.906} C_DIS
LIN {X -0.169,Y -658.893,Z 943.522,A 0.000,B 0.000,C 90.000,E1 129.930} C_DIS
LIN {X 0.256,Y -663.588,Z 943.515,A 0.000,B 0.000,C 90.000,E1 128.669} C_DIS
LIN {X 0.015,Y -670.958,Z 943.504,A 0.000,B 0.000,C 90.000,E1 126.744} C_DIS
LIN {X -0.176,Y -675.984,Z 943.496,A 0.000,B 0.000,C 90.000,E1 125.311} C_DIS
LIN {X 0.124,Y -678.403,Z 943.492,A 0.000,B 0.000,C 90.000,E1 124.565} C_DIS
LIN {X -0.109,Y -680.649,Z 943.488,A 0.000,B 0.000,C 90.000,E1 123.865} C_DIS
LIN {X -0.147,Y -684.118,Z 943.482,A 0.000,B 0.000,C 90.000,E1 122.673} C_DIS
LIN {X 0.238,Y -686.022,Z 943.478,A 0.000,B 0.000,C 90.000,E1 121.926} C_DIS
LIN {X -0.236,Y -689.313,Z 943.470,A 0.000,B 0.000,C 90.000,E1 120.541} C_DIS
LIN {X -0.172,Y -691.058,Z 943.464,A 0.000,B 0.000,C 90.000,E1 119.589} C_DIS
LIN {X 0.169,Y -692.573,Z 943.459,A 0.000,B 0.000,C 90.000,E1 118.615} C_DIS
LIN {X 0.289,Y -693.489,Z 943.455,A 0.000,B 0.000,C 90.000,E1 117.897} C_DIS
LIN {X -0.270,Y -694.401,Z 943.450,A 0.000,B 0.000,C 90.000,E1 117.001} C_DIS
LIN {X 0.113,Y -694.843,Z 943.445,A 0.000,B 0.000,C 90.000,E1 116.027} C_DIS
LIN {X 0.151,Y -695.074,Z 943.438,A 0.000,B 0.000,C 90.000,E1 114.847} C_DIS
LIN {X 0.024,Y -695.069,Z 943.436,A 0.000,B 0.000,C 90.000,E1 114.387} C_DIS
LIN {X 0.242,Y -694.840,Z 943.433,A 0.000,B 0.000,C 90.000,E1 113.898} C_DIS
LIN {X -0.173,Y -694.116,Z 943.430,A 0.000,B 0.000,C 90.000,E1 113.462} C_DIS
LIN {X 0.074,Y -693.649,Z 943.429,A 0.000,B 0.000,C 90.000,E1 113.206} C_DIS
LIN {X -0.347,Y -691.447,Z 943.426,A 0.000,B 0.000,C 90.000,E1 112.770} C_DIS
LIN {X -0.227,Y -690.860,Z 943.426,A 0.000,B 0.000,C 90.000,E1 112.642} C_DIS
LIN {X -0.109,Y -690.048,Z 943.425,A 0.000,B 0.000,C 90.000,E1 112.514} C_DIS
LIN {X 0.005,Y -688.835,Z 943.424,A 0.000,B 0.000,C 90.000,E1 112.386} C_DIS
LIN {X 0.140,Y -685.776,Z 943.423,A 0.000,B 0.000,C 90.000,E1 112.153} C_DIS
LIN {X -0.075,Y -682.743,Z 943.422,A 0.000,B 0.000,C 90.000,E1 111.972} C_DIS
LIN {X -0.312,Y -680.944,Z 943.422,A 0.000,B 0.000,C 90.000,E1 111.897} C_DIS
LIN {X -0.115,Y -676.053,Z 943.421,A 0.000,B 0.000,C 90.000,E1 111.716} C_DIS
LIN {X -0.146,Y -671.614,Z 943.420,A 0.000,B 0.000,C 90.000,E1 111.663} C_DIS
LIN {X -0.051,Y -667.641,Z 943.420,A 0.000,B 0.000,C 90.000,E1 111.589} C_DIS
LIN {X -0.229,Y -661.193,Z 943.420,A 0.000,B 0.000,C 90.000,E1 111.589} C_DIS
LIN {X -0.276,Y -636.098,Z 943.420,A 0.000,B 0.000,C 90.000,E1 111.589} C_DIS
LIN {X -0.048,Y -632.722,Z 943.420,A 0.000,B 0.000,C 90.000,E1 111.535} C_DIS
LIN {X -0.149,Y -627.065,Z 943.419,A 0.000,B 0.000,C 90.000,E1 111.461} C_DIS
LIN {X -0.046,Y -621.231,Z 943.419,A 0.000,B 0.000,C 90.000,E1 111.334} C_DIS
LIN {X 0.030,Y -615.651,Z 943.418,A 0.000,B 0.000,C 90.000,E1 111.173} C_DIS
LIN {X 0.040,Y -608.645,Z 943.416,A 0.000,B 0.000,C 90.000,E1 110.918} C_DIS
LIN {X -0.033,Y -601.826,Z 943.415,A 0.000,B 0.000,C 90.000,E1 110.610} C_DIS
LIN {X 0.236,Y -595.978,Z 943.413,A 0.000,B 0.000,C 90.000,E1 110.248} C_DIS
LIN {X -0.112,Y -587.301,Z 943.409,A 0.000,B 0.000,C 90.000,E1 109.685} C_DIS
LIN {X 0.181,Y -576.865,Z 943.405,A 0.000,B 0.000,C 90.000,E1 108.906} C_DIS
LIN {X -0.106,Y -568.361,Z 943.403,A 0.000,B 0.000,C 90.000,E1 108.471} C_DIS
LIN {X 0.116,Y -561.225,Z 943.401,A 0.000,B 0.000,C 90.000,E1 108.127} C_DIS
LIN {X 0.135,Y -553.550,Z 943.399,A 0.000,B 0.000,C 90.000,E1 107.764} C_DIS
LIN {X 0.016,Y -552.003,Z 943.398,A 0.000,B 0.000,C 90.000,E1 107.638} C_DIS
LIN {X -0.013,Y -551.974,Z 943.398,A 0.000,B 0.000,C 90.000,E1 107.638} C_DIS
LIN {X 0.113,Y -551.490,Z 943.396,A 0.000,B 0.000,C 90.000,E1 107.347} C_DIS
LIN {X -0.073,Y -551.752,Z 943.391,A 0.000,B 0.000,C 90.000,E1 106.386} C_DIS
LIN {X 0.133,Y -552.172,Z 943.385,A 0.000,B 0.000,C 90.000,E1 105.245} C_DIS
LIN {X 0.132,Y -553.279,Z 943.372,A 0.000,B 0.000,C 90.000,E1 103.008} C_DIS
LIN {X 0.055,Y -554.850,Z 943.360,A 0.000,B 0.000,C 90.000,E1 100.782} C_DIS
LIN {X 0.155,Y -556.057,Z 943.352,A 0.000,B 0.000,C 90.000,E1 99.378} C_DIS
LIN {X 0.095,Y -557.255,Z 943.344,A 0.000,B 0.000,C 90.000,E1 97.992} C_DIS
LIN {X 0.065,Y -558.357,Z 943.337,A 0.000,B 0.000,C 90.000,E1 96.606} C_DIS
LIN {X -0.081,Y -559.110,Z 943.331,A 0.000,B 0.000,C 90.000,E1 95.511} C_DIS
LIN {X -0.222,Y -559.788,Z 943.324,A 0.000,B 0.000,C 90.000,E1 94.416} C_DIS
LIN {X -0.185,Y -560.731,Z 943.315,A 0.000,B 0.000,C 90.000,E1 92.751} C_DIS
LIN {X -0.256,Y -561.345,Z 943.308,A 0.000,B 0.000,C 90.000,E1 91.375} C_DIS
LIN {X 0.234,Y -561.904,Z 943.300,A 0.000,B 0.000,C 90.000,E1 89.943} C_DIS
LIN {X 0.072,Y -562.215,Z 943.294,A 0.000,B 0.000,C 90.000,E1 88.854} C_DIS
LIN {X 0.126,Y -562.609,Z 943.285,A 0.000,B 0.000,C 90.000,E1 87.192} C_DIS
LIN {X 0.123,Y -562.851,Z 943.277,A 0.000,B 0.000,C 90.000,E1 85.812} C_DIS
LIN {X 0.131,Y -563.052,Z 943.269,A 0.000,B 0.000,C 90.000,E1 84.432} C_DIS
LIN {X 0.286,Y -563.300,Z 943.260,A 0.000,B 0.000,C 90.000,E1 82.761} C_DIS
LIN {X 0.184,Y -563.835,Z 943.248,A 0.000,B 0.000,C 90.000,E1 80.566} C_DIS
LIN {X -0.112,Y -564.389,Z 943.240,A 0.000,B 0.000,C 90.000,E1 79.218} C_DIS
LIN {X -0.115,Y -564.936,Z 943.234,A 0.000,B 0.000,C 90.000,E1 78.117} C_DIS
LIN {X 0.078,Y -566.030,Z 943.223,A 0.000,B 0.000,C 90.000,E1 76.172} C_DIS
LIN {X -0.205,Y -566.705,Z 943.217,A 0.000,B 0.000,C 90.000,E1 75.102} C_DIS
LIN {X 0.018,Y -567.710,Z 943.208,A 0.000,B 0.000,C 90.000,E1 73.433} C_DIS
LIN {X -0.244,Y -568.384,Z 943.202,A 0.000,B 0.000,C 90.000,E1 72.362} C_DIS
LIN {X 0.169,Y -569.263,Z 943.193,A 0.000,B 0.000,C 90.000,E1 70.678} C_DIS
LIN {X -0.062,Y -569.640,Z 943.188,A 0.000,B 0.000,C 90.000,E1 69.880} C_DIS
LIN {X 0.024,Y -570.184,Z 943.179,A 0.000,B 0.000,C 90.000,E1 68.230} C_DIS
LIN {X 0.149,Y -570.626,Z 943.169,A 0.000,B 0.000,C 90.000,E1 66.305} C_DIS
LIN {X 0.165,Y -570.983,Z 943.159,A 0.000,B 0.000,C 90.000,E1 64.665} C_DIS
LIN {X 0.093,Y -571.174,Z 943.152,A 0.000,B 0.000,C 90.000,E1 63.307} C_DIS
LIN {X -0.233,Y -571.301,Z 943.144,A 0.000,B 0.000,C 90.000,E1 61.975} C_DIS
LIN {X -0.080,Y -571.320,Z 943.134,A 0.000,B 0.000,C 90.000,E1 60.049} C_DIS
LIN {X 0.135,Y -571.441,Z 943.126,A 0.000,B 0.000,C 90.000,E1 58.663} C_DIS
LIN {X -0.019,Y -571.192,Z 943.117,A 0.000,B 0.000,C 90.000,E1 57.041} C_DIS
LIN {X -0.133,Y -570.851,Z 943.111,A 0.000,B 0.000,C 90.000,E1 55.960} C_DIS
LIN {X 0.193,Y -570.277,Z 943.103,A 0.000,B 0.000,C 90.000,E1 54.562} C_DIS
LIN {X -0.212,Y -569.854,Z 943.099,A 0.000,B 0.000,C 90.000,E1 53.783} C_DIS
LIN {X 0.174,Y -569.305,Z 943.094,A 0.000,B 0.000,C 90.000,E1 52.924} C_DIS
LIN {X 0.231,Y -568.296,Z 943.088,A 0.000,B 0.000,C 90.000,E1 51.823} C_DIS
LIN {X 0.157,Y -567.462,Z 943.083,A 0.000,B 0.000,C 90.000,E1 51.009} C_DIS
LIN {X 0.190,Y -566.109,Z 943.077,A 0.000,B 0.000,C 90.000,E1 49.908} C_DIS
LIN {X 0.089,Y -564.896,Z 943.073,A 0.000,B 0.000,C 90.000,E1 49.094} C_DIS
LIN {X -0.130,Y -564.051,Z 943.070,A 0.000,B 0.000,C 90.000,E1 48.566} C_DIS
LIN {X -0.210,Y -561.929,Z 943.064,A 0.000,B 0.000,C 90.000,E1 47.472} C_DIS
LIN {X -0.066,Y -560.802,Z 943.061,A 0.000,B 0.000,C 90.000,E1 46.905} C_DIS
LIN {X -0.187,Y -558.075,Z 943.054,A 0.000,B 0.000,C 90.000,E1 45.810} C_DIS
LIN {X -0.069,Y -556.590,Z 943.051,A 0.000,B 0.000,C 90.000,E1 45.243} C_DIS
LIN {X 0.041,Y -554.968,Z 943.048,A 0.000,B 0.000,C 90.000,E1 44.676} C_DIS
LIN {X -0.212,Y -552.231,Z 943.044,A 0.000,B 0.000,C 90.000,E1 43.866} C_DIS
LIN {X 0.322,Y -548.125,Z 943.037,A 0.000,B 0.000,C 90.000,E1 42.690} C_DIS
LIN {X -0.012,Y -544.551,Z 943.033,A 0.000,B 0.000,C 90.000,E1 41.881} C_DIS
LIN {X 0.045,Y -542.039,Z 943.030,A 0.000,B 0.000,C 90.000,E1 41.310} C_DIS
LIN {X 0.051,Y -536.242,Z 943.023,A 0.000,B 0.000,C 90.000,E1 40.172} C_DIS
LIN {X -0.021,Y -531.290,Z 943.018,A 0.000,B 0.000,C 90.000,E1 39.322} C_DIS
LIN {X 0.076,Y -525.258,Z 943.013,A 0.000,B 0.000,C 90.000,E1 38.302} C_DIS
LIN {X -0.173,Y -520.686,Z 943.009,A 0.000,B 0.000,C 90.000,E1 37.604} C_DIS
LIN {X 0.042,Y -516.819,Z 943.006,A 0.000,B 0.000,C 90.000,E1 36.996} C_DIS
LIN {X 0.250,Y -510.720,Z 943.001,A 0.000,B 0.000,C 90.000,E1 36.091} C_DIS
LIN {X -0.119,Y -505.296,Z 942.997,A 0.000,B 0.000,C 90.000,E1 35.391} C_DIS
LIN {X -0.126,Y -501.863,Z 942.994,A 0.000,B 0.000,C 90.000,E1 34.945} C_DIS
LIN {X 0.047,Y -496.886,Z 942.991,A 0.000,B 0.000,C 90.000,E1 34.326} C_DIS
LIN {X 0.124,Y -492.952,Z 942.988,A 0.000,B 0.000,C 90.000,E1 33.865} C_DIS
LIN {X -0.158,Y -486.179,Z 942.984,A 0.000,B 0.000,C 90.000,E1 33.166} C_DIS
LIN {X 0.105,Y -481.955,Z 942.982,A 0.000,B 0.000,C 90.000,E1 32.704} C_DIS
LIN {X 0.126,Y -474.778,Z 942.978,A 0.000,B 0.000,C 90.000,E1 32.005} C_DIS
LIN {X 0.137,Y -463.198,Z 942.972,A 0.000,B 0.000,C 90.000,E1 30.924} C_DIS
LIN {X 0.184,Y -452.617,Z 942.967,A 0.000,B 0.000,C 90.000,E1 30.001} C_DIS
LIN {X -0.043,Y -443.439,Z 942.963,A 0.000,B 0.000,C 90.000,E1 29.255} C_DIS
LIN {X -0.070,Y -429.792,Z 942.956,A 0.000,B 0.000,C 90.000,E1 28.103} C_DIS
LIN {X 0.064,Y -409.116,Z 942.946,A 0.000,B 0.000,C 90.000,E1 26.181} C_DIS
LIN {X -0.108,Y -398.897,Z 942.940,A 0.000,B 0.000,C 90.000,E1 25.155} C_DIS
LIN {X -0.002,Y -396.132,Z 942.938,A 0.000,B 0.000,C 90.000,E1 24.823} C_DIS
LIN {X 0.134,Y -392.863,Z 942.935,A 0.000,B 0.000,C 90.000,E1 24.335} C_DIS
LIN {X 0.049,Y -392.312,Z 942.935,A 0.000,B 0.000,C 90.000,E1 24.259} C_DIS
LIN {X 0.002,Y -390.525,Z 942.932,A 0.000,B 0.000,C 90.000,E1 23.823} C_DIS
LIN {X 0.212,Y -389.530,Z 942.929,A 0.000,B 0.000,C 90.000,E1 23.259} C_DIS
LIN {X -0.129,Y -389.360,Z 942.928,A 0.000,B 0.000,C 90.000,E1 23.131} C_DIS
LIN {X 0.101,Y -389.207,Z 942.924,A 0.000,B 0.000,C 90.000,E1 22.206} C_DIS
LIN {X 0.028,Y -389.853,Z 942.918,A 0.000,B 0.000,C 90.000,E1 21.153} C_DIS
LIN {X 0.058,Y -392.895,Z 942.900,A 0.000,B 0.000,C 90.000,E1 17.946} C_DIS
LIN {X -0.086,Y -396.194,Z 942.884,A 0.000,B 0.000,C 90.000,E1 15.134} C_DIS
LIN {X 0.073,Y -399.537,Z 942.870,A 0.000,B 0.000,C 90.000,E1 12.647} C_DIS
LIN {X 0.066,Y -404.417,Z 942.853,A 0.000,B 0.000,C 90.000,E1 9.500} C_DIS
LIN {X 0.113,Y -408.019,Z 942.841,A 0.000,B 0.000,C 90.000,E1 7.409} C_DIS
